  MoveL 662 to (32.13, 61.05, 0) mm, rotated rx -180 ry 0 rz -39.83 deg; joints [41.433, -75.782, 84.647, -0.866, 81.037, 41.564]
  MoveL 663 to (31.59, 62.21, 0) mm, rotated rx -180 ry 0 rz -39.83 deg; joints [41.415, -75.681, 84.52, -0.865, 81.064, 41.545]
  MoveL 664 to (31.21, 63.13, 0) mm, rotated rx 180 ry 0 rz -39.83 deg; joints [41.403, -75.601, 84.419, -0.865, 81.084, 41.533]
  MoveL 665 to (30.87, 64.05, 0) mm, rotated rx 180 ry 0 rz -39.83 deg; joints [41.392, -75.521, 84.319, -0.865, 81.105, 41.522]
  MoveL 666 to (30.56, 64.99, 0) mm, rotated rx -180 ry 0 rz -39.83 deg; joints [41.383, -75.441, 84.217, -0.865, 81.126, 41.513]
  MoveL 667 to (30.26, 65.94, 0) mm, rotated rx 180 ry 0 rz -39.83 deg; joints [41.376, -75.36, 84.115, -0.865, 81.148, 41.505]
  MoveL 668 to (30, 66.82, 0) mm, rotated rx 180 ry 0 rz -39.83 deg; joints [41.369, -75.285, 84.019, -0.865, 81.167, 41.498]
  MoveL 669 to (29.76, 67.7, 0) mm, rotated rx 180 ry 0 rz -39.83 deg; joints [41.364, -75.209, 83.924, -0.865, 81.188, 41.492]
  MoveL 670 to (29.54, 68.6, 0) mm, rotated rx 180 ry 0 rz -39.83 deg; joints [41.36, -75.134, 83.828, -0.865, 81.208, 41.488]
  MoveL 671 to (29.35, 69.49, 0) mm, rotated rx 180 ry 0 rz -39.83 deg; joints [41.357, -75.058, 83.732, -0.865, 81.228, 41.485]
  MoveL 672 to (29.18, 70.5, 0) mm, rotated rx 180 ry 0 rz -39.83 deg; joints [41.356, -74.974, 83.625, -0.865, 81.251, 41.484]
  MoveL 673 to (29.04, 71.51, 0) mm, rotated rx 180 ry 0 rz -39.83 deg; joints [41.357, -74.889, 83.518, -0.865, 81.274, 41.484]
  MoveL 674 to (28.93, 72.53, 0) mm, rotated rx 180 ry 0 rz -39.83 deg; joints [41.36, -74.805, 83.41, -0.865, 81.297, 41.487]
  MoveL 675 to (28.85, 73.55, 0) mm, rotated rx -180 ry 0 rz -39.83 deg; joints [41.364, -74.721, 83.303, -0.865, 81.32, 41.49]
  MoveL 676 to (28.8, 74.65, 0) mm, rotated rx 180 ry 0 rz -39.83 deg; joints [41.37, -74.63, 83.188, -0.865, 81.344, 41.496]
  MoveL 677 to (28.77, 75.75, 0) mm, rotated rx 180 ry 0 rz -39.83 deg; joints [41.377, -74.54, 83.073, -0.865, 81.369, 41.503]
  MoveL 678 to (28.79, 76.84, 0) mm, rotated rx 180 ry 0 rz -39.83 deg; joints [41.387, -74.45, 82.958, -0.865, 81.394, 41.512]
  MoveL 679 to (28.85, 77.94, 0) mm, rotated rx 180 ry 0 rz -39.83 deg; joints [41.399, -74.362, 82.845, -0.865, 81.419, 41.524]
  MoveL 680 to (28.94, 78.85, 0) mm, rotated rx 180 ry 0 rz -39.83 deg; joints [41.411, -74.288, 82.751, -0.865, 81.44, 41.535]
  MoveL 681 to (29.07, 79.77, 0) mm, rotated rx 180 ry 0 rz -39.83 deg; joints [41.424, -74.215, 82.657, -0.865, 81.46, 41.549]
  MoveL 682 to (29.23, 80.68, 0) mm, rotated rx 180 ry 0 rz -39.83 deg; joints [41.44, -74.142, 82.565, -0.865, 81.48, 41.564]
  MoveL 683 to (29.43, 81.58, 0) mm, rotated rx 180 ry 0 rz -39.83 deg; joints [41.457, -74.071, 82.473, -0.865, 81.501, 41.581]
  MoveL 684 to (29.67, 82.48, 0) mm, rotated rx 180 ry 0 rz -39.83 deg; joints [41.476, -74, 82.383, -0.865, 81.521, 41.6]
  MoveL 685 to (29.95, 83.36, 0) mm, rotated rx 180 ry 0 rz -39.83 deg; joints [41.498, -73.931, 82.294, -0.865, 81.54, 41.621]
  MoveL 686 to (30.28, 84.22, 0) mm, rotated rx -180 ry 0 rz -39.83 deg; joints [41.521, -73.864, 82.209, -0.865, 81.559, 41.644]
  MoveL 687 to (30.68, 85.06, 0) mm, rotated rx -180 ry 0 rz -39.83 deg; joints [41.548, -73.801, 82.128, -0.865, 81.577, 41.671]
  MoveL 688 to (30.93, 85.51, 0) mm, rotated rx 180 ry 0 rz -39.83 deg; joints [41.565, -73.767, 82.085, -0.865, 81.587, 41.687]
  MoveL 689 to (31.21, 85.95, 0) mm, rotated rx 180 ry 0 rz -39.83 deg; joints [41.582, -73.734, 82.043, -0.865, 81.596, 41.705]
  MoveL 690 to (31.51, 86.38, 0) mm, rotated rx 180 ry 0 rz -39.83 deg; joints [41.601, -73.703, 82.002, -0.865, 81.605, 41.723]
  MoveL 691 to (31.84, 86.79, 0) mm, rotated rx 180 ry 0 rz -39.83 deg; joints [41.621, -73.673, 81.964, -0.865, 81.614, 41.743]
  MoveL 692 to (32.24, 87.26, 0) mm, rotated rx 180 ry 0 rz -39.83 deg; joints [41.645, -73.639, 81.921, -0.865, 81.624, 41.767]
  MoveL 693 to (32.68, 87.7, 0) mm, rotated rx 180 ry 0 rz -39.83 deg; joints [41.671, -73.608, 81.882, -0.865, 81.632, 41.793]
  MoveL 694 to (33.15, 88.1, 0) mm, rotated rx 180 ry 0 rz -39.83 deg; joints [41.698, -73.581, 81.848, -0.865, 81.64, 41.82]
  MoveL 695 to (33.66, 88.45, 0) mm, rotated rx 180 ry 0 rz -39.83 deg; joints [41.726, -73.559, 81.819, -0.865, 81.646, 41.848]
  MoveL 696 to (33.98, 88.63, 0) mm, rotated rx 180 ry 0 rz -39.83 deg; joints [41.744, -73.547, 81.805, -0.865, 81.649, 41.866]
  MoveL 697 to (34.31, 88.8, 0) mm, rotated rx -180 ry 0 rz -39.83 deg; joints [41.762, -73.537, 81.793, -0.865, 81.652, 41.884]
  MoveL 698 to (34.64, 88.96, 0) mm, rotated rx 180 ry 0 rz -39.83 deg; joints [41.781, -73.528, 81.782, -0.865, 81.655, 41.902]
  MoveL 699 to (34.98, 89.11, 0) mm, rotated rx -180 ry 0 rz -39.83 deg; joints [41.799, -73.52, 81.771, -0.865, 81.657, 41.921]
  Establecer velocidad (1000.0 mm/s)
  MoveL 700 to (34.98, 89.11, 0) mm, rotated rx -180 ry 0 rz -39.83 deg; joints [41.799, -73.52, 81.771, -0.865, 81.657, 41.921]
  MoveL 701 to (34.98, 89.11, 20) mm, rotated rx 180 ry 0 rz -39.83 deg; joints [41.815, -73.829, 80.433, -0.862, 83.304, 41.911]

--- program P_ou_1 (robot KUKA KR 16 2) ---
  Suave(1)
  Establecer velocidad (1000.0 mm/s)
  Est. Ref.: Frame 2
  Est. herr: Plumon_ensamble
  Mostrar Plumon_ensamble
  MoveJ 1 to (24.64, 146.17, 20) mm, rotated rx 180 ry 0 rz -39.83 deg; joints [41.72, -68.932, 73.922, -0.859, 84.916, 41.792]
  MoveL 2 to (24.64, 146.17, 20) mm, rotated rx 180 ry 0 rz -39.83 deg; joints [41.72, -68.932, 73.922, -0.859, 84.916, 41.792]
  MoveL 3 to (24.64, 146.17, 0) mm, rotated rx -180 ry 0 rz -39.83 deg; joints [41.705, -68.665, 75.285, -0.861, 83.287, 41.802]
  MoveL 4 to (24.64, 146.17, 0) mm, rotated rx -180 ry 0 rz -39.83 deg; joints [41.705, -68.665, 75.285, -0.861, 83.287, 41.802]
  Establecer velocidad (50.0 mm/s)
  MoveL 5 to (24.63, 147.55, 0) mm, rotated rx 180 ry 0 rz -39.83 deg; joints [41.715, -68.548, 75.124, -0.861, 83.331, 41.811]
  MoveL 6 to (24.63, 148.94, 0) mm, rotated rx 180 ry 0 rz -39.83 deg; joints [41.724, -68.431, 74.964, -0.861, 83.375, 41.82]
  MoveL 7 to (24.65, 150.33, 0) mm, rotated rx -180 ry 0 rz -39.83 deg; joints [41.735, -68.315, 74.803, -0.861, 83.419, 41.83]
  MoveL 8 to (24.7, 151.72, 0) mm, rotated rx 180 ry 0 rz -39.83 deg; joints [41.748, -68.199, 74.643, -0.861, 83.463, 41.842]
  MoveL 9 to (24.78, 152.98, 0) mm, rotated rx 180 ry 0 rz -39.83 deg; joints [41.761, -68.093, 74.497, -0.861, 83.504, 41.854]
  MoveL 10 to (24.9, 154.25, 0) mm, rotated rx 180 ry 0 rz -39.83 deg; joints [41.775, -67.988, 74.352, -0.861, 83.544, 41.868]
  MoveL 11 to (25.06, 155.51, 0) mm, rotated rx 180 ry 0 rz -39.83 deg; joints [41.792, -67.884, 74.208, -0.861, 83.584, 41.884]
  MoveL 12 to (25.27, 156.76, 0) mm, rotated rx 180 ry 0 rz -39.83 deg; joints [41.811, -67.781, 74.065, -0.861, 83.624, 41.903]
  MoveL 13 to (25.55, 158.04, 0) mm, rotated rx 180 ry 0 rz -39.83 deg; joints [41.833, -67.676, 73.92, -0.861, 83.665, 41.924]
  MoveL 14 to (25.87, 159.31, 0) mm, rotated rx -180 ry 0 rz -39.83 deg; joints [41.858, -67.573, 73.777, -0.861, 83.705, 41.949]
  MoveL 15 to (26.26, 160.56, 0) mm, rotated rx 180 ry 0 rz -39.83 deg; joints [41.885, -67.472, 73.636, -0.861, 83.745, 41.975]
  MoveL 16 to (26.69, 161.8, 0) mm, rotated rx 180 ry 0 rz -39.83 deg; joints [41.915, -67.372, 73.498, -0.861, 83.784, 42.004]
  MoveL 17 to (27.31, 163.33, 0) mm, rotated rx 180 ry 0 rz -39.83 deg; joints [41.955, -67.25, 73.329, -0.861, 83.832, 42.043]
  MoveL 18 to (28, 164.83, 0) mm, rotated rx -180 ry 0 rz -39.83 deg; joints [41.998, -67.131, 73.163, -0.861, 83.879, 42.086]
  MoveL 19 to (28.74, 166.31, 0) mm, rotated rx -180 ry 0 rz -39.83 deg; joints [42.044, -67.014, 73, -0.861, 83.925, 42.131]
  MoveL 20 to (29.52, 167.78, 0) mm, rotated rx 180 ry 0 rz -39.83 deg; joints [42.091, -66.899, 72.84, -0.861, 83.971, 42.177]
  MoveL 21 to (30.17, 168.94, 0) mm, rotated rx -180 ry 0 rz -39.83 deg; joints [42.13, -66.807, 72.713, -0.861, 84.008, 42.216]
  MoveL 22 to (30.85, 170.09, 0) mm, rotated rx -180 ry 0 rz -39.83 deg; joints [42.17, -66.718, 72.588, -0.861, 84.043, 42.255]
  MoveL 23 to (31.58, 171.21, 0) mm, rotated rx 180 ry 0 rz -39.83 deg; joints [42.212, -66.631, 72.467, -0.861, 84.078, 42.297]
  MoveL 24 to (32.35, 172.28, 0) mm, rotated rx 180 ry 0 rz -39.83 deg; joints [42.256, -66.549, 72.352, -0.861, 84.111, 42.34]
  MoveL 25 to (33.37, 173.51, 0) mm, rotated rx 180 ry 0 rz -39.83 deg; joints [42.312, -66.456, 72.223, -0.861, 84.149, 42.396]
  MoveL 26 to (34.47, 174.67, 0) mm, rotated rx 180 ry 0 rz -39.83 deg; joints [42.372, -66.37, 72.103, -0.861, 84.184, 42.456]
  MoveL 27 to (35.63, 175.78, 0) mm, rotated rx 180 ry 0 rz -39.83 deg; joints [42.434, -66.288, 71.989, -0.861, 84.217, 42.517]
  MoveL 28 to (36.83, 176.85, 0) mm, rotated rx 180 ry 0 rz -39.83 deg; joints [42.498, -66.21, 71.88, -0.861, 84.248, 42.58]
  MoveL 29 to (38.25, 178.06, 0) mm, rotated rx 180 ry 0 rz -39.83 deg; joints [42.573, -66.123, 71.758, -0.861, 84.284, 42.655]
  MoveL 30 to (39.7, 179.21, 0) mm, rotated rx 180 ry 0 rz -39.83 deg; joints [42.649, -66.04, 71.643, -0.861, 84.317, 42.73]
  MoveL 31 to (41.21, 180.29, 0) mm, rotated rx 180 ry 0 rz -39.83 deg; joints [42.727, -65.964, 71.538, -0.861, 84.348, 42.808]
  MoveL 32 to (42.77, 181.27, 0) mm, rotated rx 180 ry 0 rz -39.83 deg; joints [42.807, -65.897, 71.445, -0.861, 84.375, 42.888]
  MoveL 33 to (43.73, 181.8, 0) mm, rotated rx -180 ry 0 rz -39.83 deg; joints [42.856, -65.863, 71.398, -0.861, 84.389, 42.936]
  MoveL 34 to (44.71, 182.29, 0) mm, rotated rx 180 ry 0 rz -39.83 deg; joints [42.905, -65.831, 71.354, -0.861, 84.402, 42.985]
  MoveL 35 to (45.7, 182.76, 0) mm, rotated rx 180 ry 0 rz -39.83 deg; joints [42.955, -65.801, 71.313, -0.861, 84.413, 43.035]
  MoveL 36 to (46.7, 183.22, 0) mm, rotated rx 180 ry 0 rz -39.83 deg; joints [43.005, -65.773, 71.274, -0.861, 84.425, 43.085]
  Establecer velocidad (1000.0 mm/s)
  MoveL 37 to (46.7, 183.22, 0) mm, rotated rx 180 ry 0 rz -39.83 deg; joints [43.005, -65.773, 71.274, -0.861, 84.425, 43.085]
  MoveL 38 to (46.7, 183.22, 20) mm, rotated rx 180 ry 0 rz -39.83 deg; joints [43.019, -66.01, 69.886, -0.859, 86.049, 43.074]
  Establecer velocidad (1000.0 mm/s)
  MoveL 39 to (24.64, 146.17, 20) mm, rotated rx 180 ry 0 rz -39.83 deg; joints [41.72, -68.932, 73.922, -0.859, 84.916, 41.792]
  MoveL 40 to (24.64, 146.17, 0) mm, rotated rx -180 ry 0 rz -39.83 deg; joints [41.705, -68.665, 75.285, -0.861, 83.287, 41.802]
  MoveL 41 to (24.64, 146.17, 0) mm, rotated rx -180 ry 0 rz -39.83 deg; joints [41.705, -68.665, 75.285, -0.861, 83.287, 41.802]
  Establecer velocidad (50.0 mm/s)
  MoveL 42 to (24.43, 145.76, 0) mm, rotated rx 180 ry 0 rz -39.83 deg; joints [41.692, -68.696, 75.328, -0.861, 83.275, 41.789]
  MoveL 43 to (24.21, 145.35, 0) mm, rotated rx 180 ry 0 rz -39.83 deg; joints [41.678, -68.728, 75.371, -0.861, 83.263, 41.776]
  MoveL 44 to (24.01, 144.94, 0) mm, rotated rx 180 ry 0 rz -39.83 deg; joints [41.666, -68.76, 75.415, -0.861, 83.252, 41.763]
  MoveL 45 to (23.83, 144.52, 0) mm, rotated rx 180 ry 0 rz -39.83 deg; joints [41.654, -68.793, 75.46, -0.861, 83.239, 41.751]
  MoveL 46 to (23.64, 144.02, 0) mm, rotated rx 180 ry 0 rz -39.83 deg; joints [41.641, -68.833, 75.513, -0.861, 83.225, 41.738]
  MoveL 47 to (23.47, 143.51, 0) mm, rotated rx 180 ry 0 rz -39.83 deg; joints [41.629, -68.873, 75.569, -0.861, 83.21, 41.727]
  MoveL 48 to (23.32, 143, 0) mm, rotated rx -180 ry 0 rz -39.83 deg; joints [41.618, -68.914, 75.625, -0.861, 83.195, 41.716]
  MoveL 49 to (23.17, 142.49, 0) mm, rotated rx 180 ry 0 rz -39.83 deg; joints [41.607, -68.955, 75.681, -0.861, 83.18, 41.705]
  MoveL 50 to (23.17, 142.49, 0) mm, rotated rx 180 ry 0 rz -39.83 deg; joints [41.607, -68.955, 75.681, -0.861, 83.18, 41.705]
  MoveL 51 to (22.09, 141.81, 0) mm, rotated rx -180 ry 0 rz -39.83 deg; joints [41.549, -68.998, 75.739, -0.861, 83.164, 41.648]
  MoveL 52 to (21.01, 141.12, 0) mm, rotated rx 180 ry 0 rz -39.83 deg; joints [41.492, -69.043, 75.798, -0.861, 83.149, 41.591]
  MoveL 53 to (19.96, 140.4, 0) mm, rotated rx 180 ry 0 rz -39.83 deg; joints [41.435, -69.09, 75.86, -0.861, 83.132, 41.534]
  MoveL 54 to (18.94, 139.64, 0) mm, rotated rx 180 ry 0 rz -39.83 deg; joints [41.38, -69.14, 75.928, -0.861, 83.114, 41.479]
  MoveL 55 to (17.59, 138.51, 0) mm, rotated rx 180 ry 0 rz -39.83 deg; joints [41.306, -69.218, 76.032, -0.861, 83.086, 41.405]
  MoveL 56 to (16.32, 137.28, 0) mm, rotated rx 180 ry 0 rz -39.83 deg; joints [41.234, -69.304, 76.149, -0.861, 83.055, 41.335]
  MoveL 57 to (15.13, 135.97, 0) mm, rotated rx 180 ry 0 rz -39.83 deg; joints [41.166, -69.398, 76.275, -0.861, 83.022, 41.267]
  MoveL 58 to (14.03, 134.58, 0) mm, rotated rx 180 ry 0 rz -39.83 deg; joints [41.102, -69.499, 76.411, -0.861, 82.986, 41.203]
  MoveL 59 to (13.16, 133.37, 0) mm, rotated rx 180 ry 0 rz -39.83 deg; joints [41.05, -69.589, 76.531, -0.861, 82.954, 41.152]
  MoveL 60 to (12.35, 132.13, 0) mm, rotated rx 180 ry 0 rz -39.83 deg; joints [41.001, -69.682, 76.657, -0.861, 82.921, 41.103]
  MoveL 61 to (11.59, 130.85, 0) mm, rotated rx 180 ry 0 rz -39.83 deg; joints [40.953, -69.778, 76.786, -0.861, 82.887, 41.056]
  MoveL 62 to (10.87, 129.55, 0) mm, rotated rx -180 ry 0 rz -39.83 deg; joints [40.908, -69.877, 76.919, -0.861, 82.853, 41.011]
  MoveL 63 to (10.02, 127.88, 0) mm, rotated rx -180 ry 0 rz -39.83 deg; joints [40.853, -70.004, 77.09, -0.861, 82.808, 40.956]
  MoveL 64 to (9.24, 126.19, 0) mm, rotated rx 180 ry 0 rz -39.83 deg; joints [40.801, -70.134, 77.265, -0.861, 82.763, 40.905]
  MoveL 65 to (8.56, 124.46, 0) mm, rotated rx 180 ry 0 rz -39.83 deg; joints [40.753, -70.269, 77.445, -0.861, 82.716, 40.858]
  MoveL 66 to (7.98, 122.69, 0) mm, rotated rx -180 ry 0 rz -39.83 deg; joints [40.71, -70.407, 77.631, -0.861, 82.668, 40.816]
  MoveL 67 to (7.57, 121.14, 0) mm, rotated rx 180 ry 0 rz -39.83 deg; joints [40.677, -70.53, 77.796, -0.861, 82.626, 40.784]
  MoveL 68 to (7.24, 119.56, 0) mm, rotated rx 180 ry 0 rz -39.83 deg; joints [40.648, -70.656, 77.964, -0.861, 82.583, 40.755]
  MoveL 69 to (6.97, 117.98, 0) mm, rotated rx -180 ry 0 rz -39.83 deg; joints [40.622, -70.784, 78.135, -0.861, 82.54, 40.73]
  MoveL 70 to (6.77, 116.38, 0) mm, rotated rx 180 ry 0 rz -39.83 deg; joints [40.598, -70.913, 78.308, -0.861, 82.496, 40.707]
  MoveL 71 to (6.61, 114.86, 0) mm, rotated rx 180 ry 0 rz -39.83 deg; joints [40.578, -71.036, 78.472, -0.861, 82.454, 40.687]
  MoveL 72 to (6.51, 113.35, 0) mm, rotated rx 180 ry 0 rz -39.83 deg; joints [40.56, -71.16, 78.637, -0.861, 82.413, 40.67]
  MoveL 73 to (6.47, 111.83, 0) mm, rotated rx -180 ry 0 rz -39.83 deg; joints [40.545, -71.285, 78.803, -0.861, 82.372, 40.655]
  MoveL 74 to (6.5, 110.32, 0) mm, rotated rx 180 ry 0 rz -39.83 deg; joints [40.534, -71.41, 78.969, -0.861, 82.33, 40.645]
  MoveL 75 to (6.61, 108.85, 0) mm, rotated rx 180 ry 0 rz -39.83 deg; joints [40.527, -71.533, 79.132, -0.861, 82.29, 40.638]
  MoveL 76 to (6.78, 107.39, 0) mm, rotated rx 180 ry 0 rz -39.83 deg; joints [40.523, -71.656, 79.295, -0.861, 82.25, 40.635]
  MoveL 77 to (7.02, 105.93, 0) mm, rotated rx -180 ry 0 rz -39.83 deg; joints [40.523, -71.779, 79.459, -0.861, 82.209, 40.636]
  MoveL 78 to (7.3, 104.48, 0) mm, rotated rx 180 ry 0 rz -39.83 deg; joints [40.525, -71.903, 79.622, -0.861, 82.17, 40.638]
  MoveL 79 to (7.53, 103.44, 0) mm, rotated rx -180 ry 0 rz -39.83 deg; joints [40.527, -71.991, 79.74, -0.861, 82.141, 40.641]
  MoveL 80 to (7.78, 102.4, 0) mm, rotated rx 180 ry 0 rz -39.83 deg; joints [40.531, -72.08, 79.857, -0.862, 82.112, 40.645]
  MoveL 81 to (8.06, 101.38, 0) mm, rotated rx 180 ry 0 rz -39.83 deg; joints [40.536, -72.168, 79.973, -0.862, 82.084, 40.651]
  MoveL 82 to (8.38, 100.36, 0) mm, rotated rx -180 ry 0 rz -39.83 deg; joints [40.543, -72.256, 80.089, -0.862, 82.056, 40.658]
  MoveL 83 to (8.85, 99.02, 0) mm, rotated rx 180 ry 0 rz -39.83 deg; joints [40.556, -72.372, 80.243, -0.862, 82.02, 40.671]
  MoveL 84 to (9.39, 97.71, 0) mm, rotated rx -180 ry 0 rz -39.83 deg; joints [40.571, -72.488, 80.395, -0.862, 81.983, 40.688]
  MoveL 85 to (9.97, 96.41, 0) mm, rotated rx 180 ry 0 rz -39.83 deg; joints [40.59, -72.603, 80.546, -0.862, 81.947, 40.707]
  MoveL 86 to (10.6, 95.12, 0) mm, rotated rx 180 ry 0 rz -39.83 deg; joints [40.61, -72.716, 80.695, -0.862, 81.912, 40.728]
  MoveL 87 to (11.22, 93.91, 0) mm, rotated rx 180 ry 0 rz -39.83 deg; joints [40.632, -72.824, 80.837, -0.862, 81.878, 40.75]
  MoveL 88 to (11.9, 92.73, 0) mm, rotated rx 180 ry 0 rz -39.83 deg; joints [40.656, -72.93, 80.976, -0.862, 81.846, 40.774]
  MoveL 89 to (12.62, 91.59, 0) mm, rotated rx 180 ry 0 rz -39.83 deg; joints [40.683, -73.034, 81.112, -0.862, 81.814, 40.802]
  MoveL 90 to (13.42, 90.49, 0) mm, rotated rx 180 ry 0 rz -39.83 deg; joints [40.714, -73.135, 81.243, -0.863, 81.783, 40.833]
  MoveL 91 to (14.09, 89.67, 0) mm, rotated rx 180 ry 0 rz -39.83 deg; joints [40.741, -73.211, 81.343, -0.863, 81.76, 40.861]
  MoveL 92 to (14.81, 88.88, 0) mm, rotated rx 180 ry 0 rz -39.83 deg; joints [40.771, -73.285, 81.44, -0.863, 81.737, 40.891]
  MoveL 93 to (15.55, 88.11, 0) mm, rotated rx 180 ry 0 rz -39.83 deg; joints [40.802, -73.358, 81.536, -0.863, 81.715, 40.922]
  MoveL 94 to (16.3, 87.35, 0) mm, rotated rx 180 ry 0 rz -39.83 deg; joints [40.833, -73.43, 81.63, -0.863, 81.694, 40.954]
  MoveL 95 to (16.3, 87.35, 0) mm, rotated rx 180 ry 0 rz -39.83 deg; joints [40.833, -73.43, 81.63, -0.863, 81.694, 40.954]
  MoveL 96 to (16.8, 85.15, 0) mm, rotated rx 180 ry 0 rz -39.83 deg; joints [40.841, -73.617, 81.872, -0.863, 81.638, 40.962]
  MoveL 97 to (17.32, 82.96, 0) mm, rotated rx -180 ry 0 rz -39.83 deg; joints [40.849, -73.803, 82.113, -0.863, 81.584, 40.971]
  MoveL 98 to (17.9, 80.78, 0) mm, rotated rx 180 ry 0 rz -39.83 deg; joints [40.86, -73.989, 82.353, -0.863, 81.53, 40.983]
  MoveL 99 to (18.54, 78.63, 0) mm, rotated rx 180 ry 0 rz -39.83 deg; joints [40.875, -74.174, 82.591, -0.864, 81.477, 40.999]
  MoveL 100 to (19.22, 76.65, 0) mm, rotated rx 180 ry 0 rz -39.83 deg; joints [40.893, -74.345, 82.811, -0.864, 81.429, 41.018]
  MoveL 101 to (19.97, 74.68, 0) mm, rotated rx 180 ry 0 rz -39.83 deg; joints [40.915, -74.515, 83.029, -0.864, 81.381, 41.04]
  MoveL 102 to (20.75, 72.73, 0) mm, rotated rx 180 ry 0 rz -39.83 deg; joints [40.939, -74.684, 83.246, -0.864, 81.334, 41.065]
  MoveL 103 to (21.56, 70.79, 0) mm, rotated rx 180 ry 0 rz -39.83 deg; joints [40.964, -74.854, 83.462, -0.864, 81.287, 41.091]
  MoveL 104 to (21.56, 70.79, 0) mm, rotated rx 180 ry 0 rz -39.83 deg; joints [40.964, -74.854, 83.462, -0.864, 81.287, 41.091]
  MoveL 105 to (22.1, 68.18, 0) mm, rotated rx 180 ry 0 rz -39.83 deg; joints [40.971, -75.074, 83.742, -0.864, 81.228, 41.098]
  MoveL 106 to (22.69, 65.58, 0) mm, rotated rx -180 ry 0 rz -39.83 deg; joints [40.979, -75.294, 84.021, -0.864, 81.169, 41.108]
  MoveL 107 to (23.37, 63, 0) mm, rotated rx 180 ry 0 rz -39.83 deg; joints [40.993, -75.512, 84.297, -0.865, 81.111, 41.122]
  MoveL 108 to (24.17, 60.46, 0) mm, rotated rx 180 ry 0 rz -39.83 deg; joints [41.013, -75.729, 84.571, -0.865, 81.055, 41.144]
  MoveL 109 to (24.64, 59.19, 0) mm, rotated rx -180 ry 0 rz -39.83 deg; joints [41.027, -75.839, 84.709, -0.865, 81.027, 41.158]
  MoveL 110 to (25.16, 57.94, 0) mm, rotated rx 180 ry 0 rz -39.83 deg; joints [41.044, -75.948, 84.846, -0.865, 80.999, 41.175]
  MoveL 111 to (25.74, 56.72, 0) mm, rotated rx 180 ry 0 rz -39.83 deg; joints [41.064, -76.055, 84.98, -0.865, 80.972, 41.196]
  MoveL 112 to (26.38, 55.53, 0) mm, rotated rx -180 ry 0 rz -39.83 deg; joints [41.088, -76.16, 85.112, -0.865, 80.945, 41.22]
  MoveL 113 to (27.01, 54.5, 0) mm, rotated rx 180 ry 0 rz -39.83 deg; joints [41.112, -76.252, 85.228, -0.865, 80.922, 41.245]
  MoveL 114 to (27.68, 53.5, 0) mm, rotated rx 180 ry 0 rz -39.83 deg; joints [41.139, -76.342, 85.341, -0.865, 80.899, 41.272]
  MoveL 115 to (28.39, 52.51, 0) mm, rotated rx 180 ry 0 rz -39.83 deg; joints [41.168, -76.431, 85.453, -0.866, 80.877, 41.301]
  MoveL 116 to (29.11, 51.54, 0) mm, rotated rx 180 ry 0 rz -39.83 deg; joints [41.197, -76.52, 85.564, -0.866, 80.855, 41.331]
  MoveL 117 to (29.89, 50.49, 0) mm, rotated rx 180 ry 0 rz -39.83 deg; joints [41.23, -76.614, 85.682, -0.866, 80.832, 41.364]
  MoveL 118 to (30.7, 49.47, 0) mm, rotated rx -180 ry 0 rz -39.83 deg; joints [41.264, -76.708, 85.799, -0.866, 80.809, 41.398]
  MoveL 119 to (31.53, 48.46, 0) mm, rotated rx 180 ry 0 rz -39.83 deg; joints [41.299, -76.8, 85.914, -0.866, 80.787, 41.434]
  MoveL 120 to (32.39, 47.49, 0) mm, rotated rx 180 ry 0 rz -39.83 deg; joints [41.337, -76.891, 86.027, -0.866, 80.765, 41.472]
  MoveL 121 to (33.11, 46.72, 0) mm, rotated rx 180 ry 0 rz -39.83 deg; joints [41.369, -76.962, 86.116, -0.866, 80.748, 41.504]
  MoveL 122 to (33.87, 45.98, 0) mm, rotated rx -180 ry 0 rz -39.83 deg; joints [41.403, -77.031, 86.202, -0.866, 80.731, 41.539]
  MoveL 123 to (34.65, 45.27, 0) mm, rotated rx -180 ry 0 rz -39.83 deg; joints [41.439, -77.098, 86.286, -0.866, 80.715, 41.574]
  MoveL 124 to (35.45, 44.59, 0) mm, rotated rx 180 ry 0 rz -39.83 deg; joints [41.476, -77.164, 86.368, -0.866, 80.7, 41.612]
  MoveL 125 to (36.39, 43.86, 0) mm, rotated rx 180 ry 0 rz -39.83 deg; joints [41.52, -77.235, 86.456, -0.867, 80.683, 41.656]
  MoveL 126 to (37.35, 43.16, 0) mm, rotated rx -180 ry 0 rz -39.83 deg; joints [41.565, -77.303, 86.542, -0.867, 80.667, 41.702]
  MoveL 127 to (38.33, 42.49, 0) mm, rotated rx 180 ry 0 rz -39.83 deg; joints [41.612, -77.37, 86.625, -0.867, 80.651, 41.749]
  MoveL 128 to (39.32, 41.83, 0) mm, rotated rx 180 ry 0 rz -39.83 deg; joints [41.659, -77.435, 86.706, -0.867, 80.635, 41.797]
  MoveL 129 to (40.09, 41.34, 0) mm, rotated rx 180 ry 0 rz -39.83 deg; joints [41.696, -77.484, 86.767, -0.867, 80.624, 41.834]
  MoveL 130 to (40.86, 40.86, 0) mm, rotated rx -180 ry 0 rz -39.83 deg; joints [41.733, -77.533, 86.827, -0.867, 80.613, 41.871]
  MoveL 131 to (41.64, 40.4, 0) mm, rotated rx 180 ry 0 rz -39.83 deg; joints [41.771, -77.579, 86.886, -0.867, 80.602, 41.909]
  MoveL 132 to (42.43, 39.96, 0) mm, rotated rx -180 ry 0 rz -39.83 deg; joints [41.81, -77.624, 86.942, -0.867, 80.591, 41.948]
  MoveL 133 to (43.59, 39.38, 0) mm, rotated rx 180 ry 0 rz -39.83 deg; joints [41.867, -77.685, 87.017, -0.867, 80.577, 42.006]
  MoveL 134 to (44.76, 38.84, 0) mm, rotated rx 180 ry 0 rz -39.83 deg; joints [41.926, -77.743, 87.089, -0.868, 80.564, 42.065]
  MoveL 135 to (45.96, 38.33, 0) mm, rotated rx 180 ry 0 rz -39.83 deg; joints [41.986, -77.798, 87.158, -0.868, 80.551, 42.125]
  MoveL 136 to (47.15, 37.83, 0) mm, rotated rx 180 ry 0 rz -39.83 deg; joints [42.047, -77.852, 87.226, -0.868, 80.539, 42.185]
  MoveL 137 to (47.15, 37.83, 0) mm, rotated rx 180 ry 0 rz -39.83 deg; joints [42.047, -77.852, 87.226, -0.868, 80.539, 42.185]
  MoveL 138 to (48.32, 36.91, 0) mm, rotated rx 180 ry 0 rz -39.83 deg; joints [42.102, -77.941, 87.335, -0.868, 80.519, 42.241]
  MoveL 139 to (49.49, 35.99, 0) mm, rotated rx 180 ry 0 rz -39.83 deg; joints [42.158, -78.029, 87.443, -0.868, 80.499, 42.297]
  MoveL 140 to (50.68, 35.09, 0) mm, rotated rx -180 ry 0 rz -39.83 deg; joints [42.215, -78.115, 87.55, -0.868, 80.48, 42.355]
  MoveL 141 to (51.89, 34.23, 0) mm, rotated rx -180 ry 0 rz -39.83 deg; joints [42.273, -78.199, 87.653, -0.868, 80.461, 42.413]
  MoveL 142 to (52.71, 33.66, 0) mm, rotated rx 180 ry 0 rz -39.83 deg; joints [42.314, -78.254, 87.721, -0.868, 80.449, 42.454]
  MoveL 143 to (53.55, 33.11, 0) mm, rotated rx 180 ry 0 rz -39.83 deg; joints [42.355, -78.308, 87.788, -0.869, 80.437, 42.495]
  MoveL 144 to (54.4, 32.58, 0) mm, rotated rx -180 ry 0 rz -39.83 deg; joints [42.397, -78.361, 87.853, -0.869, 80.426, 42.537]
  MoveL 145 to (55.26, 32.05, 0) mm, rotated rx 180 ry 0 rz -39.83 deg; joints [42.439, -78.413, 87.917, -0.869, 80.414, 42.58]
  MoveL 146 to (56.32, 31.41, 0) mm, rotated rx -180 ry 0 rz -39.83 deg; joints [42.492, -78.477, 87.995, -0.869, 80.401, 42.633]
  MoveL 147 to (57.4, 30.78, 0) mm, rotated rx 180 ry 0 rz -39.83 deg; joints [42.545, -78.54, 88.072, -0.869, 80.387, 42.686]
  MoveL 148 to (58.48, 30.17, 0) mm, rotated rx 180 ry 0 rz -39.83 deg; joints [42.599, -78.601, 88.148, -0.869, 80.374, 42.741]
  MoveL 149 to (59.57, 29.58, 0) mm, rotated rx 180 ry 0 rz -39.83 deg; joints [42.654, -78.661, 88.221, -0.869, 80.361, 42.796]
  MoveL 150 to (60.92, 28.87, 0) mm, rotated rx -180 ry 0 rz -39.83 deg; joints [42.723, -78.732, 88.309, -0.869, 80.346, 42.865]
  MoveL 151 to (62.29, 28.2, 0) mm, rotated rx 180 ry 0 rz -39.83 deg; joints [42.792, -78.802, 88.394, -0.869, 80.331, 42.934]
  MoveL 152 to (63.68, 27.55, 0) mm, rotated rx 180 ry 0 rz -39.83 deg; joints [42.863, -78.869, 88.476, -0.87, 80.317, 43.005]
  MoveL 153 to (65.07, 26.93, 0) mm, rotated rx 180 ry 0 rz -39.83 deg; joints [42.934, -78.933, 88.556, -0.87, 80.303, 43.077]
  MoveL 154 to (66.63, 26.27, 0) mm, rotated rx -180 ry 0 rz -39.83 deg; joints [43.015, -79.003, 88.641, -0.87, 80.289, 43.158]
  MoveL 155 to (68.2, 25.64, 0) mm, rotated rx 180 ry 0 rz -39.83 deg; joints [43.096, -79.07, 88.724, -0.87, 80.274, 43.239]
  MoveL 156 to (69.78, 25.02, 0) mm, rotated rx 180 ry 0 rz -39.83 deg; joints [43.177, -79.136, 88.805, -0.87, 80.261, 43.321]
  MoveL 157 to (71.36, 24.41, 0) mm, rotated rx 180 ry 0 rz -39.83 deg; joints [43.259, -79.201, 88.885, -0.87, 80.247, 43.403]
  MoveL 158 to (71.36, 24.41, 0) mm, rotated rx 180 ry 0 rz -39.83 deg; joints [43.259, -79.201, 88.885, -0.87, 80.247, 43.403]
  MoveL 159 to (71.89, 23.71, 0) mm, rotated rx -180 ry 0 rz -39.83 deg; joints [43.284, -79.264, 88.96, -0.87, 80.235, 43.428]
  MoveL 160 to (72.42, 23.01, 0) mm, rotated rx 180 ry 0 rz -39.83 deg; joints [43.309, -79.326, 89.034, -0.87, 80.222, 43.453]
  MoveL 161 to (72.98, 22.34, 0) mm, rotated rx 180 ry 0 rz -39.83 deg; joints [43.335, -79.386, 89.107, -0.87, 80.211, 43.479]
  MoveL 162 to (73.57, 21.7, 0) mm, rotated rx 180 ry 0 rz -39.83 deg; joints [43.363, -79.444, 89.177, -0.871, 80.199, 43.507]
  MoveL 163 to (74.45, 20.85, 0) mm, rotated rx 180 ry 0 rz -39.83 deg; joints [43.406, -79.521, 89.27, -0.871, 80.184, 43.55]
  MoveL 164 to (75.39, 20.07, 0) mm, rotated rx 180 ry 0 rz -39.83 deg; joints [43.452, -79.594, 89.357, -0.871, 80.17, 43.597]
  MoveL 165 to (76.37, 19.33, 0) mm, rotated rx 180 ry 0 rz -39.83 deg; joints [43.501, -79.663, 89.441, -0.871, 80.156, 43.646]
  MoveL 166 to (77.37, 18.62, 0) mm, rotated rx 180 ry 0 rz -39.83 deg; joints [43.551, -79.731, 89.522, -0.871, 80.143, 43.697]
  MoveL 167 to (78.43, 17.9, 0) mm, rotated rx 180 ry 0 rz -39.83 deg; joints [43.605, -79.8, 89.605, -0.871, 80.13, 43.75]
  MoveL 168 to (79.49, 17.19, 0) mm, rotated rx -180 ry 0 rz -39.83 deg; joints [43.658, -79.867, 89.686, -0.871, 80.117, 43.804]
  MoveL 169 to (80.56, 16.5, 0) mm, rotated rx 180 ry 0 rz -39.83 deg; joints [43.713, -79.933, 89.765, -0.871, 80.105, 43.859]
  MoveL 170 to (81.65, 15.85, 0) mm, rotated rx 180 ry 0 rz -39.83 deg; joints [43.769, -79.996, 89.842, -0.871, 80.093, 43.915]
  MoveL 171 to (82.83, 15.18, 0) mm, rotated rx -180 ry 0 rz -39.83 deg; joints [43.83, -80.061, 89.92, -0.871, 80.08, 43.977]
  MoveL 172 to (84.04, 14.56, 0) mm, rotated rx 180 ry 0 rz -39.83 deg; joints [43.893, -80.123, 89.994, -0.872, 80.069, 44.04]
  MoveL 173 to (85.27, 13.98, 0) mm, rotated rx -180 ry 0 rz -39.83 deg; joints [43.958, -80.18, 90.064, -0.872, 80.058, 44.104]
  MoveL 174 to (86.52, 13.46, 0) mm, rotated rx -180 ry 0 rz -39.83 deg; joints [44.024, -80.234, 90.128, -0.872, 80.048, 44.171]
  MoveL 175 to (87.55, 13.07, 0) mm, rotated rx 180 ry 0 rz -39.83 deg; joints [44.078, -80.274, 90.177, -0.872, 80.04, 44.226]
  MoveL 176 to (88.59, 12.73, 0) mm, rotated rx -180 ry 0 rz -39.83 deg; joints [44.134, -80.311, 90.222, -0.872, 80.033, 44.281]
  MoveL 177 to (89.64, 12.42, 0) mm, rotated rx 180 ry 0 rz -39.83 deg; joints [44.191, -80.346, 90.263, -0.872, 80.027, 44.338]
  MoveL 178 to (90.7, 12.13, 0) mm, rotated rx 180 ry 0 rz -39.83 deg; joints [44.248, -80.377, 90.302, -0.872, 80.02, 44.395]
  MoveL 179 to (91.93, 11.85, 0) mm, rotated rx -180 ry 0 rz -39.83 deg; joints [44.314, -80.411, 90.343, -0.872, 80.014, 44.462]
  MoveL 180 to (93.17, 11.59, 0) mm, rotated rx 180 ry 0 rz -39.83 deg; joints [44.382, -80.442, 90.381, -0.872, 80.008, 44.529]
  MoveL 181 to (94.41, 11.38, 0) mm, rotated rx 180 ry 0 rz -39.83 deg; joints [44.449, -80.469, 90.415, -0.872, 80.003, 44.597]
  MoveL 182 to (95.66, 11.19, 0) mm, rotated rx 180 ry 0 rz -39.83 deg; joints [44.518, -80.494, 90.445, -0.872, 79.998, 44.666]
  MoveL 183 to (96.8, 11.06, 0) mm, rotated rx 180 ry 0 rz -39.83 deg; joints [44.58, -80.514, 90.47, -0.872, 79.994, 44.728]
  MoveL 184 to (97.94, 10.95, 0) mm, rotated rx 180 ry 0 rz -39.83 deg; joints [44.643, -80.532, 90.492, -0.872, 79.99, 44.791]
  MoveL 185 to (99.09, 10.88, 0) mm, rotated rx 180 ry 0 rz -39.83 deg; joints [44.706, -80.546, 90.511, -0.873, 79.987, 44.855]
  MoveL 186 to (100.23, 10.85, 0) mm, rotated rx 180 ry 0 rz -39.83 deg; joints [44.77, -80.557, 90.525, -0.873, 79.985, 44.918]
  MoveL 187 to (100.6, 10.85, 0) mm, rotated rx 180 ry 0 rz -39.83 deg; joints [44.79, -80.56, 90.529, -0.873, 79.984, 44.939]
  MoveL 188 to (100.96, 10.86, 0) mm, rotated rx 180 ry 0 rz -39.83 deg; joints [44.811, -80.562, 90.532, -0.873, 79.984, 44.959]
  MoveL 189 to (101.33, 10.87, 0) mm, rotated rx -180 ry 0 rz -39.83 deg; joints [44.831, -80.564, 90.535, -0.873, 79.983, 44.979]
  MoveL 190 to (101.69, 10.88, 0) mm, rotated rx 180 ry 0 rz -39.83 deg; joints [44.851, -80.565, 90.537, -0.873, 79.983, 45]
  MoveL 191 to (101.69, 10.88, 0) mm, rotated rx 180 ry 0 rz -39.83 deg; joints [44.851, -80.565, 90.537, -0.873, 79.983, 45]
  MoveL 192 to (102.06, 10.87, 0) mm, rotated rx 180 ry 0 rz -39.83 deg; joints [44.872, -80.569, 90.542, -0.873, 79.982, 45.02]
  MoveL 193 to (102.43, 10.86, 0) mm, rotated rx 180 ry 0 rz -39.83 deg; joints [44.892, -80.573, 90.546, -0.873, 79.981, 45.04]
  MoveL 194 to (102.79, 10.85, 0) mm, rotated rx 180 ry 0 rz -39.83 deg; joints [44.912, -80.576, 90.55, -0.873, 79.98, 45.061]
  MoveL 195 to (103.16, 10.85, 0) mm, rotated rx 180 ry 0 rz -39.83 deg; joints [44.933, -80.578, 90.554, -0.873, 79.98, 45.081]
  MoveL 196 to (104.3, 10.88, 0) mm, rotated rx 180 ry 0 rz -39.83 deg; joints [44.997, -80.584, 90.562, -0.873, 79.978, 45.145]
  MoveL 197 to (105.45, 10.95, 0) mm, rotated rx -180 ry 0 rz -39.83 deg; joints [45.061, -80.587, 90.567, -0.873, 79.977, 45.209]
  MoveL 198 to (106.59, 11.06, 0) mm, rotated rx 180 ry 0 rz -39.83 deg; joints [45.125, -80.586, 90.568, -0.873, 79.977, 45.273]
  MoveL 199 to (107.73, 11.19, 0) mm, rotated rx 180 ry 0 rz -39.83 deg; joints [45.189, -80.583, 90.565, -0.873, 79.977, 45.337]
  MoveL 200 to (108.98, 11.38, 0) mm, rotated rx -180 ry 0 rz -39.83 deg; joints [45.259, -80.576, 90.559, -0.873, 79.977, 45.408]
  MoveL 201 to (110.22, 11.59, 0) mm, rotated rx 180 ry 0 rz -39.83 deg; joints [45.33, -80.567, 90.55, -0.873, 79.978, 45.478]
  MoveL 202 to (111.46, 11.85, 0) mm, rotated rx -180 ry 0 rz -39.83 deg; joints [45.4, -80.554, 90.537, -0.873, 79.98, 45.548]
  MoveL 203 to (112.68, 12.13, 0) mm, rotated rx 180 ry 0 rz -39.83 deg; joints [45.469, -80.539, 90.52, -0.873, 79.982, 45.618]
  MoveL 204 to (113.75, 12.42, 0) mm, rotated rx 180 ry 0 rz -39.83 deg; joints [45.53, -80.522, 90.502, -0.873, 79.984, 45.678]
  MoveL 205 to (114.8, 12.73, 0) mm, rotated rx 180 ry 0 rz -39.83 deg; joints [45.59, -80.503, 90.482, -0.873, 79.987, 45.738]
  MoveL 206 to (115.84, 13.07, 0) mm, rotated rx 180 ry 0 rz -39.83 deg; joints [45.649, -80.482, 90.457, -0.873, 79.99, 45.798]
  MoveL 207 to (116.87, 13.46, 0) mm, rotated rx 180 ry 0 rz -39.83 deg; joints [45.708, -80.457, 90.429, -0.873, 79.994, 45.856]
  MoveL 208 to (118.12, 13.98, 0) mm, rotated rx 180 ry 0 rz -39.83 deg; joints [45.78, -80.421, 90.39, -0.873, 80, 45.928]
  MoveL 209 to (119.35, 14.56, 0) mm, rotated rx 180 ry 0 rz -39.83 deg; joints [45.851, -80.381, 90.344, -0.873, 80.006, 45.999]
  MoveL 210 to (120.56, 15.18, 0) mm, rotated rx 180 ry 0 rz -39.83 deg; joints [45.921, -80.337, 90.294, -0.873, 80.013, 46.069]
  MoveL 211 to (121.74, 15.85, 0) mm, rotated rx 180 ry 0 rz -39.83 deg; joints [45.989, -80.289, 90.24, -0.873, 80.021, 46.137]
  MoveL 212 to (122.83, 16.5, 0) mm, rotated rx -180 ry 0 rz -39.83 deg; joints [46.052, -80.242, 90.185, -0.873, 80.029, 46.2]
  MoveL 213 to (123.9, 17.19, 0) mm, rotated rx 180 ry 0 rz -39.83 deg; joints [46.114, -80.191, 90.127, -0.873, 80.037, 46.262]
  MoveL 214 to (124.96, 17.9, 0) mm, rotated rx 180 ry 0 rz -39.83 deg; joints [46.176, -80.139, 90.067, -0.873, 80.046, 46.324]
  MoveL 215 to (126.01, 18.62, 0) mm, rotated rx -180 ry 0 rz -39.83 deg; joints [46.237, -80.085, 90.005, -0.873, 80.055, 46.384]
  MoveL 216 to (127.02, 19.33, 0) mm, rotated rx -180 ry 0 rz -39.83 deg; joints [46.295, -80.032, 89.944, -0.873, 80.064, 46.443]
  MoveL 217 to (128, 20.07, 0) mm, rotated rx -180 ry 0 rz -39.83 deg; joints [46.352, -79.977, 89.88, -0.873, 80.074, 46.499]
  MoveL 218 to (128.94, 20.85, 0) mm, rotated rx 180 ry 0 rz -39.83 deg; joints [46.407, -79.917, 89.811, -0.873, 80.084, 46.554]
  MoveL 219 to (129.82, 21.7, 0) mm, rotated rx 180 ry 0 rz -39.83 deg; joints [46.459, -79.853, 89.736, -0.873, 80.095, 46.606]
  MoveL 220 to (130.4, 22.34, 0) mm, rotated rx 180 ry 0 rz -39.83 deg; joints [46.494, -79.803, 89.678, -0.873, 80.104, 46.64]
  MoveL 221 to (130.96, 23.01, 0) mm, rotated rx 180 ry 0 rz -39.83 deg; joints [46.527, -79.75, 89.616, -0.873, 80.114, 46.674]
  MoveL 222 to (131.5, 23.71, 0) mm, rotated rx -180 ry 0 rz -39.83 deg; joints [46.559, -79.696, 89.553, -0.873, 80.123, 46.706]
  MoveL 223 to (132.03, 24.41, 0) mm, rotated rx 180 ry 0 rz -39.83 deg; joints [46.591, -79.641, 89.488, -0.873, 80.133, 46.737]
  MoveL 224 to (132.03, 24.41, 0) mm, rotated rx 180 ry 0 rz -39.83 deg; joints [46.591, -79.641, 89.488, -0.873, 80.133, 46.737]
  MoveL 225 to (133.61, 25.02, 0) mm, rotated rx 180 ry 0 rz -39.83 deg; joints [46.68, -79.599, 89.44, -0.873, 80.141, 46.826]
  MoveL 226 to (135.19, 25.64, 0) mm, rotated rx 180 ry 0 rz -39.83 deg; joints [46.769, -79.555, 89.39, -0.873, 80.148, 46.915]
  MoveL 227 to (136.75, 26.27, 0) mm, rotated rx 180 ry 0 rz -39.83 deg; joints [46.857, -79.51, 89.339, -0.873, 80.156, 47.003]
  MoveL 228 to (138.31, 26.93, 0) mm, rotated rx 180 ry 0 rz -39.83 deg; joints [46.945, -79.463, 89.284, -0.873, 80.164, 47.091]
  MoveL 229 to (139.71, 27.55, 0) mm, rotated rx 180 ry 0 rz -39.83 deg; joints [47.024, -79.418, 89.233, -0.873, 80.172, 47.17]
  MoveL 230 to (141.09, 28.2, 0) mm, rotated rx 180 ry 0 rz -39.83 deg; joints [47.102, -79.371, 89.178, -0.873, 80.18, 47.248]
  MoveL 231 to (142.46, 28.87, 0) mm, rotated rx -180 ry 0 rz -39.83 deg; joints [47.18, -79.321, 89.121, -0.873, 80.189, 47.325]
  MoveL 232 to (143.82, 29.58, 0) mm, rotated rx 180 ry 0 rz -39.83 deg; joints [47.256, -79.268, 89.06, -0.873, 80.199, 47.402]
  MoveL 233 to (144.91, 30.17, 0) mm, rotated rx 180 ry 0 rz -39.83 deg; joints [47.318, -79.224, 89.008, -0.873, 80.207, 47.463]
  MoveL 234 to (145.99, 30.78, 0) mm, rotated rx 180 ry 0 rz -39.83 deg; joints [47.379, -79.178, 88.955, -0.873, 80.215, 47.524]
  MoveL 235 to (147.07, 31.41, 0) mm, rotated rx 180 ry 0 rz -39.83 deg; joints [47.439, -79.13, 88.899, -0.873, 80.224, 47.584]
  MoveL 236 to (148.13, 32.05, 0) mm, rotated rx -180 ry 0 rz -39.83 deg; joints [47.5, -79.081, 88.842, -0.873, 80.233, 47.644]
  MoveL 237 to (148.99, 32.58, 0) mm, rotated rx 180 ry 0 rz -39.83 deg; joints [47.548, -79.041, 88.795, -0.873, 80.24, 47.693]
  MoveL 238 to (149.83, 33.11, 0) mm, rotated rx 180 ry 0 rz -39.83 deg; joints [47.596, -79, 88.747, -0.873, 80.248, 47.74]
  MoveL 239 to (150.67, 33.66, 0) mm, rotated rx -180 ry 0 rz -39.83 deg; joints [47.643, -78.958, 88.698, -0.873, 80.256, 47.788]
  MoveL 240 to (151.5, 34.23, 0) mm, rotated rx 180 ry 0 rz -39.83 deg; joints [47.69, -78.914, 88.647, -0.873, 80.264, 47.834]
  MoveL 241 to (152.71, 35.09, 0) mm, rotated rx 180 ry 0 rz -39.83 deg; joints [47.758, -78.847, 88.567, -0.873, 80.277, 47.902]
  MoveL 242 to (153.9, 35.99, 0) mm, rotated rx 180 ry 0 rz -39.83 deg; joints [47.825, -78.777, 88.485, -0.873, 80.291, 47.969]
  MoveL 243 to (155.07, 36.91, 0) mm, rotated rx 180 ry 0 rz -39.83 deg; joints [47.891, -78.705, 88.4, -0.873, 80.305, 48.035]
  MoveL 244 to (156.23, 37.83, 0) mm, rotated rx 180 ry 0 rz -39.83 deg; joints [47.956, -78.633, 88.314, -0.873, 80.319, 48.1]
  MoveL 245 to (156.23, 37.83, 0) mm, rotated rx 180 ry 0 rz -39.83 deg; joints [47.956, -78.633, 88.314, -0.873, 80.319, 48.1]
  MoveL 246 to (157.43, 38.33, 0) mm, rotated rx 180 ry 0 rz -39.83 deg; joints [48.023, -78.595, 88.271, -0.873, 80.326, 48.167]
  MoveL 247 to (158.63, 38.84, 0) mm, rotated rx 180 ry 0 rz -39.83 deg; joints [48.089, -78.557, 88.226, -0.873, 80.333, 48.232]
  MoveL 248 to (159.8, 39.38, 0) mm, rotated rx 180 ry 0 rz -39.83 deg; joints [48.154, -78.515, 88.178, -0.873, 80.341, 48.298]
  MoveL 249 to (160.96, 39.96, 0) mm, rotated rx 180 ry 0 rz -39.83 deg; joints [48.218, -78.471, 88.125, -0.873, 80.35, 48.362]
  MoveL 250 to (161.75, 40.4, 0) mm, rotated rx -180 ry 0 rz -39.83 deg; joints [48.262, -78.437, 88.085, -0.873, 80.357, 48.405]
  MoveL 251 to (162.53, 40.86, 0) mm, rotated rx 180 ry 0 rz -39.83 deg; joints [48.306, -78.4, 88.043, -0.873, 80.364, 48.449]
  MoveL 252 to (163.3, 41.34, 0) mm, rotated rx -180 ry 0 rz -39.83 deg; joints [48.348, -78.363, 87.998, -0.873, 80.371, 48.491]
  MoveL 253 to (164.06, 41.83, 0) mm, rotated rx 180 ry 0 rz -39.83 deg; joints [48.391, -78.324, 87.953, -0.873, 80.379, 48.534]
  MoveL 254 to (165.06, 42.49, 0) mm, rotated rx 180 ry 0 rz -39.83 deg; joints [48.446, -78.273, 87.891, -0.873, 80.389, 48.589]
  MoveL 255 to (166.04, 43.16, 0) mm, rotated rx 180 ry 0 rz -39.83 deg; joints [48.5, -78.219, 87.828, -0.873, 80.4, 48.643]
  MoveL 256 to (167, 43.86, 0) mm, rotated rx 180 ry 0 rz -39.83 deg; joints [48.554, -78.164, 87.762, -0.873, 80.411, 48.696]
  MoveL 257 to (167.94, 44.59, 0) mm, rotated rx 180 ry 0 rz -39.83 deg; joints [48.606, -78.105, 87.692, -0.873, 80.423, 48.748]
  MoveL 258 to (168.74, 45.27, 0) mm, rotated rx -180 ry 0 rz -39.83 deg; joints [48.65, -78.051, 87.628, -0.873, 80.435, 48.792]
  MoveL 259 to (169.52, 45.98, 0) mm, rotated rx 180 ry 0 rz -39.83 deg; joints [48.694, -77.994, 87.559, -0.873, 80.447, 48.835]
  MoveL 260 to (170.27, 46.72, 0) mm, rotated rx 180 ry 0 rz -39.83 deg; joints [48.736, -77.935, 87.488, -0.873, 80.459, 48.877]
  MoveL 261 to (171, 47.49, 0) mm, rotated rx -180 ry 0 rz -39.83 deg; joints [48.776, -77.873, 87.414, -0.873, 80.472, 48.917]
  MoveL 262 to (171.86, 48.46, 0) mm, rotated rx 180 ry 0 rz -39.83 deg; joints [48.824, -77.794, 87.32, -0.873, 80.489, 48.965]
  MoveL 263 to (172.69, 49.47, 0) mm, rotated rx -180 ry 0 rz -39.83 deg; joints [48.87, -77.713, 87.221, -0.872, 80.506, 49.011]
  MoveL 264 to (173.49, 50.49, 0) mm, rotated rx 180 ry 0 rz -39.83 deg; joints [48.915, -77.63, 87.121, -0.872, 80.524, 49.055]
  MoveL 265 to (174.28, 51.54, 0) mm, rotated rx 180 ry 0 rz -39.83 deg; joints [48.958, -77.545, 87.019, -0.872, 80.543, 49.098]
  MoveL 266 to (175, 52.51, 0) mm, rotated rx -180 ry 0 rz -39.83 deg; joints [48.998, -77.466, 86.923, -0.872, 80.56, 49.138]
  MoveL 267 to (175.7, 53.5, 0) mm, rotated rx 180 ry 0 rz -39.83 deg; joints [49.037, -77.386, 86.825, -0.872, 80.578, 49.177]
  MoveL 268 to (176.38, 54.5, 0) mm, rotated rx 180 ry 0 rz -39.83 deg; joints [49.074, -77.304, 86.726, -0.872, 80.596, 49.214]
  MoveL 269 to (177, 55.53, 0) mm, rotated rx 180 ry 0 rz -39.83 deg; joints [49.109, -77.22, 86.624, -0.872, 80.615, 49.248]
  MoveL 270 to (177.65, 56.72, 0) mm, rotated rx -180 ry 0 rz -39.83 deg; joints [49.145, -77.123, 86.505, -0.872, 80.637, 49.284]
  MoveL 271 to (178.22, 57.94, 0) mm, rotated rx -180 ry 0 rz -39.83 deg; joints [49.177, -77.023, 86.383, -0.872, 80.66, 49.315]
  MoveL 272 to (178.75, 59.19, 0) mm, rotated rx 180 ry 0 rz -39.83 deg; joints [49.206, -76.921, 86.257, -0.872, 80.683, 49.344]
  MoveL 273 to (179.22, 60.46, 0) mm, rotated rx 180 ry 0 rz -39.83 deg; joints [49.232, -76.817, 86.129, -0.872, 80.707, 49.37]
  MoveL 274 to (180.02, 63, 0) mm, rotated rx 180 ry 0 rz -39.83 deg; joints [49.278, -76.609, 85.873, -0.872, 80.757, 49.415]
  MoveL 275 to (180.7, 65.58, 0) mm, rotated rx -180 ry 0 rz -39.83 deg; joints [49.316, -76.397, 85.611, -0.872, 80.807, 49.452]
  MoveL 276 to (181.29, 68.18, 0) mm, rotated rx -180 ry 0 rz -39.83 deg; joints [49.349, -76.184, 85.346, -0.871, 80.859, 49.485]
  MoveL 277 to (181.83, 70.79, 0) mm, rotated rx 180 ry 0 rz -39.83 deg; joints [49.38, -75.969, 85.079, -0.871, 80.913, 49.515]
  MoveL 278 to (181.83, 70.79, 0) mm, rotated rx 180 ry 0 rz -39.83 deg; joints [49.38, -75.969, 85.079, -0.871, 80.913, 49.515]
  MoveL 279 to (182.64, 72.73, 0) mm, rotated rx 180 ry 0 rz -39.83 deg; joints [49.424, -75.81, 84.88, -0.871, 80.952, 49.558]
  MoveL 280 to (183.42, 74.68, 0) mm, rotated rx 180 ry 0 rz -39.83 deg; joints [49.467, -75.649, 84.68, -0.871, 80.993, 49.6]
  MoveL 281 to (184.16, 76.65, 0) mm, rotated rx 180 ry 0 rz -39.83 deg; joints [49.507, -75.488, 84.478, -0.871, 81.034, 49.64]
  MoveL 282 to (184.84, 78.63, 0) mm, rotated rx -180 ry 0 rz -39.83 deg; joints [49.544, -75.325, 84.273, -0.871, 81.076, 49.676]
  MoveL 283 to (185.49, 80.78, 0) mm, rotated rx -180 ry 0 rz -39.83 deg; joints [49.579, -75.147, 84.049, -0.871, 81.123, 49.711]
  MoveL 284 to (186.06, 82.96, 0) mm, rotated rx 180 ry 0 rz -39.83 deg; joints [49.611, -74.968, 83.823, -0.871, 81.17, 49.741]
  MoveL 285 to (186.59, 85.15, 0) mm, rotated rx 180 ry 0 rz -39.83 deg; joints [49.639, -74.787, 83.594, -0.87, 81.219, 49.769]
  MoveL 286 to (187.09, 87.35, 0) mm, rotated rx -180 ry 0 rz -39.83 deg; joints [49.667, -74.605, 83.363, -0.87, 81.268, 49.796]
  MoveL 287 to (187.09, 87.35, 0) mm, rotated rx -180 ry 0 rz -39.83 deg; joints [49.667, -74.605, 83.363, -0.87, 81.268, 49.796]
  MoveL 288 to (187.84, 88.11, 0) mm, rotated rx 180 ry 0 rz -39.83 deg; joints [49.706, -74.543, 83.285, -0.87, 81.285, 49.835]
  MoveL 289 to (188.58, 88.88, 0) mm, rotated rx 180 ry 0 rz -39.83 deg; joints [49.745, -74.479, 83.205, -0.87, 81.302, 49.874]
  MoveL 290 to (189.29, 89.67, 0) mm, rotated rx 180 ry 0 rz -39.83 deg; joints [49.782, -74.414, 83.123, -0.87, 81.319, 49.911]
  MoveL 291 to (189.97, 90.49, 0) mm, rotated rx 180 ry 0 rz -39.83 deg; joints [49.818, -74.347, 83.038, -0.87, 81.338, 49.946]
  MoveL 292 to (190.77, 91.59, 0) mm, rotated rx 180 ry 0 rz -39.83 deg; joints [49.86, -74.256, 82.923, -0.87, 81.363, 49.987]
  MoveL 293 to (191.49, 92.73, 0) mm, rotated rx 180 ry 0 rz -39.83 deg; joints [49.898, -74.162, 82.803, -0.87, 81.389, 50.025]
  MoveL 294 to (192.16, 93.91, 0) mm, rotated rx -180 ry 0 rz -39.83 deg; joints [49.933, -74.064, 82.678, -0.87, 81.416, 50.06]
  MoveL 295 to (192.79, 95.12, 0) mm, rotated rx 180 ry 0 rz -39.83 deg; joints [49.966, -73.964, 82.55, -0.87, 81.444, 50.092]
  MoveL 296 to (193.42, 96.41, 0) mm, rotated rx -180 ry 0 rz -39.83 deg; joints [49.998, -73.858, 82.415, -0.87, 81.474, 50.124]
  MoveL 297 to (194, 97.71, 0) mm, rotated rx 180 ry 0 rz -39.83 deg; joints [50.029, -73.75, 82.277, -0.87, 81.505, 50.154]
  MoveL 298 to (194.54, 99.02, 0) mm, rotated rx 180 ry 0 rz -39.83 deg; joints [50.057, -73.641, 82.137, -0.87, 81.536, 50.182]
  MoveL 299 to (195.01, 100.36, 0) mm, rotated rx 180 ry 0 rz -39.83 deg; joints [50.081, -73.53, 81.994, -0.869, 81.569, 50.206]
  MoveL 300 to (195.32, 101.38, 0) mm, rotated rx 180 ry 0 rz -39.83 deg; joints [50.097, -73.446, 81.885, -0.869, 81.593, 50.222]
  MoveL 301 to (195.6, 102.4, 0) mm, rotated rx -180 ry 0 rz -39.83 deg; joints [50.112, -73.361, 81.776, -0.869, 81.618, 50.236]
  MoveL 302 to (195.86, 103.44, 0) mm, rotated rx 180 ry 0 rz -39.83 deg; joints [50.125, -73.275, 81.665, -0.869, 81.643, 50.248]
  MoveL 303 to (196.09, 104.48, 0) mm, rotated rx 180 ry 0 rz -39.83 deg; joints [50.137, -73.188, 81.553, -0.869, 81.669, 50.26]
  MoveL 304 to (196.37, 105.93, 0) mm, rotated rx 180 ry 0 rz -39.83 deg; joints [50.151, -73.068, 81.396, -0.869, 81.705, 50.274]
  MoveL 305 to (196.61, 107.39, 0) mm, rotated rx 180 ry 0 rz -39.83 deg; joints [50.164, -72.947, 81.239, -0.869, 81.741, 50.285]
  MoveL 306 to (196.78, 108.85, 0) mm, rotated rx -180 ry 0 rz -39.83 deg; joints [50.173, -72.825, 81.081, -0.869, 81.778, 50.294]
  MoveL 307 to (196.89, 110.32, 0) mm, rotated rx 180 ry 0 rz -39.83 deg; joints [50.178, -72.703, 80.922, -0.869, 81.815, 50.299]
  MoveL 308 to (196.92, 111.83, 0) mm, rotated rx -180 ry 0 rz -39.83 deg; joints [50.18, -72.577, 80.757, -0.869, 81.854, 50.3]
  MoveL 309 to (196.88, 113.35, 0) mm, rotated rx -180 ry 0 rz -39.83 deg; joints [50.178, -72.451, 80.592, -0.869, 81.893, 50.297]
  MoveL 310 to (196.78, 114.86, 0) mm, rotated rx 180 ry 0 rz -39.83 deg; joints [50.172, -72.325, 80.426, -0.869, 81.932, 50.291]
  MoveL 311 to (196.62, 116.38, 0) mm, rotated rx 180 ry 0 rz -39.83 deg; joints [50.164, -72.199, 80.26, -0.869, 81.972, 50.283]
  MoveL 312 to (196.41, 117.98, 0) mm, rotated rx 180 ry 0 rz -39.83 deg; joints [50.154, -72.066, 80.085, -0.868, 82.014, 50.272]
  MoveL 313 to (196.15, 119.56, 0) mm, rotated rx -180 ry 0 rz -39.83 deg; joints [50.141, -71.933, 79.91, -0.868, 82.057, 50.258]
  MoveL 314 to (195.82, 121.14, 0) mm, rotated rx -180 ry 0 rz -39.83 deg; joints [50.124, -71.802, 79.737, -0.868, 82.099, 50.24]
  MoveL 315 to (195.41, 122.69, 0) mm, rotated rx 180 ry 0 rz -39.83 deg; joints [50.103, -71.673, 79.565, -0.868, 82.141, 50.219]
  MoveL 316 to (194.83, 124.46, 0) mm, rotated rx -180 ry 0 rz -39.83 deg; joints [50.074, -71.525, 79.369, -0.868, 82.189, 50.189]
  MoveL 317 to (194.14, 126.19, 0) mm, rotated rx -180 ry 0 rz -39.83 deg; joints [50.04, -71.381, 79.176, -0.868, 82.237, 50.154]
  MoveL 318 to (193.37, 127.88, 0) mm, rotated rx 180 ry 0 rz -39.83 deg; joints [50.001, -71.239, 78.986, -0.868, 82.284, 50.114]
  MoveL 319 to (192.52, 129.55, 0) mm, rotated rx 180 ry 0 rz -39.83 deg; joints [49.958, -71.1, 78.8, -0.868, 82.331, 50.071]
  MoveL 320 to (191.8, 130.85, 0) mm, rotated rx -180 ry 0 rz -39.83 deg; joints [49.922, -70.991, 78.653, -0.868, 82.368, 50.035]
  MoveL 321 to (191.04, 132.13, 0) mm, rotated rx 180 ry 0 rz -39.83 deg; joints [49.884, -70.884, 78.509, -0.868, 82.404, 49.996]
  MoveL 322 to (190.23, 133.37, 0) mm, rotated rx 180 ry 0 rz -39.83 deg; joints [49.844, -70.779, 78.368, -0.868, 82.44, 49.955]
  MoveL 323 to (189.36, 134.58, 0) mm, rotated rx 180 ry 0 rz -39.83 deg; joints [49.801, -70.677, 78.231, -0.868, 82.475, 49.912]
  MoveL 324 to (188.26, 135.97, 0) mm, rotated rx 180 ry 0 rz -39.83 deg; joints [49.746, -70.561, 78.074, -0.868, 82.515, 49.856]
  MoveL 325 to (187.07, 137.28, 0) mm, rotated rx -180 ry 0 rz -39.83 deg; joints [49.688, -70.451, 77.923, -0.868, 82.554, 49.797]
  MoveL 326 to (185.8, 138.51, 0) mm, rotated rx 180 ry 0 rz -39.83 deg; joints [49.625, -70.347, 77.782, -0.868, 82.59, 49.734]
  MoveL 327 to (184.45, 139.64, 0) mm, rotated rx 180 ry 0 rz -39.83 deg; joints [49.558, -70.25, 77.651, -0.867, 82.624, 49.666]
  MoveL 328 to (183.43, 140.4, 0) mm, rotated rx -180 ry 0 rz -39.83 deg; joints [49.508, -70.186, 77.562, -0.867, 82.648, 49.616]
  MoveL 329 to (182.37, 141.12, 0) mm, rotated rx -180 ry 0 rz -39.83 deg; joints [49.456, -70.125, 77.478, -0.867, 82.669, 49.563]
  MoveL 330 to (181.3, 141.81, 0) mm, rotated rx 180 ry 0 rz -39.83 deg; joints [49.403, -70.066, 77.398, -0.867, 82.691, 49.51]
  MoveL 331 to (180.22, 142.49, 0) mm, rotated rx -180 ry 0 rz -39.83 deg; joints [49.349, -70.008, 77.318, -0.867, 82.712, 49.456]
  MoveL 332 to (180.22, 142.49, 0) mm, rotated rx -180 ry 0 rz -39.83 deg; joints [49.349, -70.008, 77.318, -0.867, 82.712, 49.456]
  MoveL 333 to (180.07, 143, 0) mm, rotated rx 180 ry 0 rz -39.83 deg; joints [49.342, -69.965, 77.259, -0.867, 82.727, 49.449]
  MoveL 334 to (179.92, 143.51, 0) mm, rotated rx 180 ry 0 rz -39.83 deg; joints [49.335, -69.921, 77.2, -0.867, 82.742, 49.442]
  MoveL 335 to (179.75, 144.02, 0) mm, rotated rx -180 ry 0 rz -39.83 deg; joints [49.327, -69.879, 77.142, -0.867, 82.758, 49.434]
  MoveL 336 to (179.56, 144.52, 0) mm, rotated rx -180 ry 0 rz -39.83 deg; joints [49.318, -69.837, 77.085, -0.867, 82.773, 49.424]
  MoveL 337 to (179.38, 144.94, 0) mm, rotated rx 180 ry 0 rz -39.83 deg; joints [49.309, -69.801, 77.037, -0.867, 82.785, 49.415]
  MoveL 338 to (179.17, 145.35, 0) mm, rotated rx 180 ry 0 rz -39.83 deg; joints [49.3, -69.766, 76.989, -0.867, 82.798, 49.405]
  MoveL 339 to (178.96, 145.76, 0) mm, rotated rx -180 ry 0 rz -39.83 deg; joints [49.289, -69.731, 76.942, -0.867, 82.81, 49.395]
  MoveL 340 to (178.74, 146.17, 0) mm, rotated rx 180 ry 0 rz -39.83 deg; joints [49.279, -69.697, 76.894, -0.867, 82.823, 49.384]
  MoveL 341 to (178.74, 146.17, 0) mm, rotated rx 180 ry 0 rz -39.83 deg; joints [49.279, -69.697, 76.894, -0.867, 82.823, 49.384]
  MoveL 342 to (178.76, 147.55, 0) mm, rotated rx 180 ry 0 rz -39.83 deg; joints [49.281, -69.58, 76.736, -0.867, 82.865, 49.385]
  MoveL 343 to (178.76, 148.94, 0) mm, rotated rx -180 ry 0 rz -39.83 deg; joints [49.282, -69.463, 76.576, -0.867, 82.907, 49.386]
  MoveL 344 to (178.74, 150.33, 0) mm, rotated rx 180 ry 0 rz -39.83 deg; joints [49.282, -69.346, 76.417, -0.867, 82.949, 49.385]
  MoveL 345 to (178.69, 151.72, 0) mm, rotated rx -180 ry 0 rz -39.83 deg; joints [49.281, -69.228, 76.257, -0.867, 82.992, 49.383]
  MoveL 346 to (178.61, 152.98, 0) mm, rotated rx 180 ry 0 rz -39.83 deg; joints [49.278, -69.121, 76.111, -0.867, 83.031, 49.38]
  MoveL 347 to (178.49, 154.25, 0) mm, rotated rx 180 ry 0 rz -39.83 deg; joints [49.273, -69.014, 75.965, -0.867, 83.07, 49.374]
  MoveL 348 to (178.33, 155.51, 0) mm, rotated rx 180 ry 0 rz -39.83 deg; joints [49.266, -68.908, 75.818, -0.867, 83.11, 49.367]
  MoveL 349 to (178.11, 156.76, 0) mm, rotated rx 180 ry 0 rz -39.83 deg; joints [49.256, -68.802, 75.673, -0.867, 83.149, 49.356]
  MoveL 350 to (177.84, 158.04, 0) mm, rotated rx 180 ry 0 rz -39.83 deg; joints [49.244, -68.693, 75.523, -0.867, 83.19, 49.343]
  MoveL 351 to (177.51, 159.31, 0) mm, rotated rx -180 ry 0 rz -39.83 deg; joints [49.229, -68.585, 75.374, -0.866, 83.23, 49.328]
  MoveL 352 to (177.13, 160.56, 0) mm, rotated rx -180 ry 0 rz -39.83 deg; joints [49.211, -68.478, 75.227, -0.866, 83.271, 49.31]
  MoveL 353 to (176.7, 161.8, 0) mm, rotated rx 180 ry 0 rz -39.83 deg; joints [49.191, -68.373, 75.081, -0.866, 83.311, 49.289]
  MoveL 354 to (176.08, 163.33, 0) mm, rotated rx 180 ry 0 rz -39.83 deg; joints [49.162, -68.242, 74.9, -0.866, 83.361, 49.259]
  MoveL 355 to (175.39, 164.83, 0) mm, rotated rx -180 ry 0 rz -39.83 deg; joints [49.13, -68.113, 74.721, -0.866, 83.41, 49.226]
  MoveL 356 to (174.65, 166.31, 0) mm, rotated rx 180 ry 0 rz -39.83 deg; joints [49.095, -67.986, 74.544, -0.866, 83.459, 49.19]
  MoveL 357 to (173.87, 167.78, 0) mm, rotated rx 180 ry 0 rz -39.83 deg; joints [49.058, -67.861, 74.369, -0.866, 83.508, 49.153]
  MoveL 358 to (173.21, 168.94, 0) mm, rotated rx -180 ry 0 rz -39.83 deg; joints [49.028, -67.76, 74.229, -0.866, 83.548, 49.122]
  MoveL 359 to (172.53, 170.09, 0) mm, rotated rx -180 ry 0 rz -39.83 deg; joints [48.996, -67.661, 74.091, -0.866, 83.586, 49.089]
  MoveL 360 to (171.81, 171.21, 0) mm, rotated rx 180 ry 0 rz -39.83 deg; joints [48.962, -67.565, 73.956, -0.866, 83.624, 49.055]
  MoveL 361 to (171.03, 172.28, 0) mm, rotated rx 180 ry 0 rz -39.83 deg; joints [48.925, -67.472, 73.826, -0.866, 83.661, 49.018]
  MoveL 362 to (170.01, 173.51, 0) mm, rotated rx 180 ry 0 rz -39.83 deg; joints [48.877, -67.366, 73.676, -0.866, 83.704, 48.969]
  MoveL 363 to (168.92, 174.67, 0) mm, rotated rx 180 ry 0 rz -39.83 deg; joints [48.825, -67.265, 73.534, -0.866, 83.744, 48.917]
  MoveL 364 to (167.76, 175.78, 0) mm, rotated rx 180 ry 0 rz -39.83 deg; joints [48.771, -67.168, 73.397, -0.866, 83.784, 48.861]
  MoveL 365 to (166.56, 176.85, 0) mm, rotated rx 180 ry 0 rz -39.83 deg; joints [48.714, -67.073, 73.263, -0.866, 83.822, 48.804]
  MoveL 366 to (165.14, 178.06, 0) mm, rotated rx 180 ry 0 rz -39.83 deg; joints [48.647, -66.967, 73.112, -0.866, 83.865, 48.737]
  MoveL 367 to (163.69, 179.21, 0) mm, rotated rx 180 ry 0 rz -39.83 deg; joints [48.579, -66.865, 72.967, -0.865, 83.907, 48.668]
  MoveL 368 to (162.18, 180.29, 0) mm, rotated rx 180 ry 0 rz -39.83 deg; joints [48.508, -66.769, 72.831, -0.865, 83.947, 48.596]
  MoveL 369 to (160.62, 181.27, 0) mm, rotated rx 180 ry 0 rz -39.83 deg; joints [48.434, -66.681, 72.705, -0.865, 83.983, 48.522]
  MoveL 370 to (159.66, 181.8, 0) mm, rotated rx 180 ry 0 rz -39.83 deg; joints [48.389, -66.634, 72.638, -0.865, 84.003, 48.476]
  MoveL 371 to (158.68, 182.29, 0) mm, rotated rx 180 ry 0 rz -39.83 deg; joints [48.342, -66.589, 72.574, -0.865, 84.022, 48.429]
  MoveL 372 to (157.68, 182.76, 0) mm, rotated rx 180 ry 0 rz -39.83 deg; joints [48.295, -66.546, 72.512, -0.865, 84.04, 48.382]
  MoveL 373 to (156.68, 183.22, 0) mm, rotated rx 180 ry 0 rz -39.83 deg; joints [48.248, -66.504, 72.451, -0.865, 84.058, 48.335]
  MoveL 374 to (156.68, 183.22, 0) mm, rotated rx 180 ry 0 rz -39.83 deg; joints [48.248, -66.504, 72.451, -0.865, 84.058, 48.335]
  MoveL 375 to (156.82, 183.34, 0) mm, rotated rx 180 ry 0 rz -39.83 deg; joints [48.255, -66.494, 72.437, -0.865, 84.062, 48.341]
  MoveL 376 to (156.96, 183.47, 0) mm, rotated rx 180 ry 0 rz -39.83 deg; joints [48.262, -66.484, 72.422, -0.865, 84.066, 48.348]
  MoveL 377 to (157.11, 183.58, 0) mm, rotated rx 180 ry 0 rz -39.83 deg; joints [48.269, -66.474, 72.409, -0.865, 84.07, 48.356]
  MoveL 378 to (157.26, 183.68, 0) mm, rotated rx 180 ry 0 rz -39.83 deg; joints [48.277, -66.466, 72.398, -0.865, 84.073, 48.363]
  MoveL 379 to (157.57, 183.82, 0) mm, rotated rx -180 ry 0 rz -39.83 deg; joints [48.292, -66.455, 72.383, -0.865, 84.077, 48.378]
  MoveL 380 to (157.9, 183.91, 0) mm, rotated rx -180 ry 0 rz -39.83 deg; joints [48.308, -66.448, 72.373, -0.865, 84.08, 48.394]
  MoveL 381 to (158.24, 183.98, 0) mm, rotated rx 180 ry 0 rz -39.83 deg; joints [48.324, -66.442, 72.366, -0.865, 84.082, 48.41]
  MoveL 382 to (158.58, 184.05, 0) mm, rotated rx 180 ry 0 rz -39.83 deg; joints [48.341, -66.438, 72.36, -0.865, 84.084, 48.427]
  MoveL 383 to (159.29, 184.23, 0) mm, rotated rx 180 ry 0 rz -39.83 deg; joints [48.375, -66.424, 72.342, -0.865, 84.089, 48.461]
  MoveL 384 to (159.97, 184.45, 0) mm, rotated rx -180 ry 0 rz -39.83 deg; joints [48.408, -66.406, 72.317, -0.865, 84.096, 48.494]
  MoveL 385 to (160.64, 184.71, 0) mm, rotated rx 180 ry 0 rz -39.83 deg; joints [48.44, -66.386, 72.29, -0.865, 84.104, 48.526]
  MoveL 386 to (161.32, 184.97, 0) mm, rotated rx 180 ry 0 rz -39.83 deg; joints [48.473, -66.365, 72.261, -0.865, 84.112, 48.559]
  MoveL 387 to (161.8, 185.16, 0) mm, rotated rx 180 ry 0 rz -39.83 deg; joints [48.496, -66.35, 72.241, -0.865, 84.118, 48.582]
  MoveL 388 to (162.28, 185.35, 0) mm, rotated rx 180 ry 0 rz -39.83 deg; joints [48.52, -66.335, 72.22, -0.865, 84.124, 48.605]
  MoveL 389 to (162.75, 185.57, 0) mm, rotated rx 180 ry 0 rz -39.83 deg; joints [48.542, -66.317, 72.195, -0.865, 84.131, 48.628]
  MoveL 390 to (163.18, 185.83, 0) mm, rotated rx 180 ry 0 rz -39.83 deg; joints [48.564, -66.295, 72.165, -0.865, 84.14, 48.649]
  MoveL 391 to (163.55, 186.12, 0) mm, rotated rx 180 ry 0 rz -39.83 deg; joints [48.582, -66.271, 72.131, -0.865, 84.149, 48.667]
  MoveL 392 to (163.89, 186.45, 0) mm, rotated rx 180 ry 0 rz -39.83 deg; joints [48.598, -66.243, 72.093, -0.865, 84.161, 48.683]
  MoveL 393 to (164.2, 186.81, 0) mm, rotated rx -180 ry 0 rz -39.83 deg; joints [48.613, -66.213, 72.05, -0.865, 84.173, 48.698]
  MoveL 394 to (164.48, 187.19, 0) mm, rotated rx 180 ry 0 rz -39.83 deg; joints [48.627, -66.181, 72.005, -0.865, 84.186, 48.712]
  MoveL 395 to (164.68, 187.5, 0) mm, rotated rx 180 ry 0 rz -39.83 deg; joints [48.637, -66.155, 71.969, -0.865, 84.197, 48.721]
  MoveL 396 to (164.86, 187.81, 0) mm, rotated rx 180 ry 0 rz -39.83 deg; joints [48.646, -66.128, 71.931, -0.865, 84.208, 48.73]
  MoveL 397 to (165.02, 188.14, 0) mm, rotated rx 180 ry 0 rz -39.83 deg; joints [48.654, -66.101, 71.892, -0.865, 84.219, 48.738]
  MoveL 398 to (165.16, 188.47, 0) mm, rotated rx 180 ry 0 rz -39.83 deg; joints [48.662, -66.072, 71.852, -0.865, 84.231, 48.746]
  MoveL 399 to (165.23, 188.65, 0) mm, rotated rx 180 ry 0 rz -39.83 deg; joints [48.665, -66.057, 71.831, -0.865, 84.237, 48.749]
  MoveL 400 to (165.28, 188.82, 0) mm, rotated rx 180 ry 0 rz -39.83 deg; joints [48.668, -66.042, 71.809, -0.865, 84.243, 48.751]
  MoveL 401 to (165.32, 189, 0) mm, rotated rx 180 ry 0 rz -39.83 deg; joints [48.67, -66.026, 71.788, -0.865, 84.25, 48.754]
  MoveL 402 to (165.35, 189.18, 0) mm, rotated rx 180 ry 0 rz -39.83 deg; joints [48.671, -66.011, 71.766, -0.865, 84.256, 48.755]
  MoveL 403 to (165.36, 189.35, 0) mm, rotated rx 180 ry 0 rz -39.83 deg; joints [48.672, -65.996, 71.745, -0.865, 84.262, 48.755]
  MoveL 404 to (165.35, 189.53, 0) mm, rotated rx -180 ry 0 rz -39.83 deg; joints [48.672, -65.981, 71.724, -0.865, 84.269, 48.755]
  MoveL 405 to (165.33, 189.7, 0) mm, rotated rx 180 ry 0 rz -39.83 deg; joints [48.671, -65.966, 71.703, -0.865, 84.275, 48.754]
  MoveL 406 to (165.31, 189.87, 0) mm, rotated rx 180 ry 0 rz -39.83 deg; joints [48.67, -65.952, 71.682, -0.865, 84.281, 48.753]
  MoveL 407 to (165.31, 189.87, 0) mm, rotated rx 180 ry 0 rz -39.83 deg; joints [48.67, -65.952, 71.682, -0.865, 84.281, 48.753]
  MoveL 408 to (166.15, 190.18, 0) mm, rotated rx 180 ry 0 rz -39.83 deg; joints [48.711, -65.926, 71.647, -0.865, 84.291, 48.794]
  MoveL 409 to (166.99, 190.51, 0) mm, rotated rx 180 ry 0 rz -39.83 deg; joints [48.751, -65.9, 71.611, -0.865, 84.302, 48.834]
  MoveL 410 to (167.81, 190.85, 0) mm, rotated rx 180 ry 0 rz -39.83 deg; joints [48.791, -65.872, 71.571, -0.865, 84.313, 48.874]
  MoveL 411 to (168.62, 191.24, 0) mm, rotated rx 180 ry 0 rz -39.83 deg; joints [48.83, -65.84, 71.528, -0.865, 84.326, 48.912]
  MoveL 412 to (169.24, 191.57, 0) mm, rotated rx 180 ry 0 rz -39.83 deg; joints [48.86, -65.812, 71.489, -0.865, 84.337, 48.942]
  MoveL 413 to (169.84, 191.94, 0) mm, rotated rx 180 ry 0 rz -39.83 deg; joints [48.889, -65.781, 71.446, -0.865, 84.35, 48.971]
  MoveL 414 to (170.42, 192.34, 0) mm, rotated rx 180 ry 0 rz -39.83 deg; joints [48.917, -65.748, 71.399, -0.865, 84.363, 48.999]
  MoveL 415 to (170.97, 192.78, 0) mm, rotated rx -180 ry 0 rz -39.83 deg; joints [48.944, -65.71, 71.347, -0.865, 84.379, 49.025]
  MoveL 416 to (171.39, 193.17, 0) mm, rotated rx 180 ry 0 rz -39.83 deg; joints [48.964, -65.678, 71.301, -0.865, 84.392, 49.045]
  MoveL 417 to (171.78, 193.58, 0) mm, rotated rx 180 ry 0 rz -39.83 deg; joints [48.983, -65.643, 71.251, -0.865, 84.407, 49.064]
  MoveL 418 to (172.14, 194.03, 0) mm, rotated rx -180 ry 0 rz -39.83 deg; joints [49, -65.605, 71.198, -0.865, 84.423, 49.081]
  MoveL 419 to (172.44, 194.5, 0) mm, rotated rx -180 ry 0 rz -39.83 deg; joints [49.015, -65.564, 71.14, -0.865, 84.44, 49.096]
  MoveL 420 to (172.6, 194.81, 0) mm, rotated rx 180 ry 0 rz -39.83 deg; joints [49.023, -65.537, 71.103, -0.865, 84.451, 49.103]
  MoveL 421 to (172.73, 195.13, 0) mm, rotated rx 180 ry 0 rz -39.83 deg; joints [49.03, -65.51, 71.064, -0.865, 84.463, 49.11]
  MoveL 422 to (172.85, 195.46, 0) mm, rotated rx 180 ry 0 rz -39.83 deg; joints [49.036, -65.482, 71.024, -0.865, 84.474, 49.116]
  MoveL 423 to (172.95, 195.79, 0) mm, rotated rx 180 ry 0 rz -39.83 deg; joints [49.04, -65.453, 70.983, -0.864, 84.487, 49.12]
  MoveL 424 to (173.04, 196.19, 0) mm, rotated rx -180 ry 0 rz -39.83 deg; joints [49.045, -65.418, 70.934, -0.864, 84.501, 49.125]
  MoveL 425 to (173.1, 196.59, 0) mm, rotated rx 180 ry 0 rz -39.83 deg; joints [49.049, -65.384, 70.884, -0.864, 84.516, 49.128]
  MoveL 426 to (173.16, 197, 0) mm, rotated rx 180 ry 0 rz -39.83 deg; joints [49.052, -65.349, 70.834, -0.864, 84.531, 49.131]
  MoveL 427 to (173.2, 197.4, 0) mm, rotated rx 180 ry 0 rz -39.83 deg; joints [49.054, -65.314, 70.784, -0.864, 84.546, 49.133]
  MoveL 428 to (173.2, 197.4, 0) mm, rotated rx 180 ry 0 rz -39.83 deg; joints [49.054, -65.314, 70.784, -0.864, 84.546, 49.133]
  MoveL 429 to (173.89, 197.88, 0) mm, rotated rx 180 ry 0 rz -39.83 deg; joints [49.087, -65.273, 70.727, -0.864, 84.563, 49.166]
  MoveL 430 to (174.56, 198.37, 0) mm, rotated rx -180 ry 0 rz -39.83 deg; joints [49.12, -65.232, 70.669, -0.864, 84.58, 49.198]
  MoveL 431 to (175.23, 198.87, 0) mm, rotated rx 180 ry 0 rz -39.83 deg; joints [49.152, -65.189, 70.61, -0.864, 84.598, 49.23]
  MoveL 432 to (175.88, 199.38, 0) mm, rotated rx 180 ry 0 rz -39.83 deg; joints [49.183, -65.145, 70.548, -0.864, 84.616, 49.261]
  MoveL 433 to (176.34, 199.76, 0) mm, rotated rx 180 ry 0 rz -39.83 deg; joints [49.205, -65.113, 70.502, -0.864, 84.63, 49.282]
  MoveL 434 to (176.78, 200.15, 0) mm, rotated rx 180 ry 0 rz -39.83 deg; joints [49.226, -65.08, 70.455, -0.864, 84.644, 49.303]
  MoveL 435 to (177.21, 200.55, 0) mm, rotated rx -180 ry 0 rz -39.83 deg; joints [49.247, -65.046, 70.407, -0.864, 84.659, 49.324]
  MoveL 436 to (177.65, 200.95, 0) mm, rotated rx -180 ry 0 rz -39.83 deg; joints [49.268, -65.011, 70.358, -0.864, 84.673, 49.345]
  MoveL 437 to (178.02, 201.32, 0) mm, rotated rx 180 ry 0 rz -39.83 deg; joints [49.286, -64.98, 70.313, -0.864, 84.687, 49.363]
  MoveL 438 to (178.38, 201.7, 0) mm, rotated rx -180 ry 0 rz -39.83 deg; joints [49.303, -64.947, 70.267, -0.864, 84.7, 49.38]
  MoveL 439 to (178.71, 202.1, 0) mm, rotated rx -180 ry 0 rz -39.83 deg; joints [49.319, -64.913, 70.218, -0.864, 84.715, 49.395]
  MoveL 440 to (178.99, 202.53, 0) mm, rotated rx 180 ry 0 rz -39.83 deg; joints [49.332, -64.876, 70.165, -0.864, 84.731, 49.408]
  MoveL 441 to (179.14, 202.84, 0) mm, rotated rx 180 ry 0 rz -39.83 deg; joints [49.34, -64.848, 70.126, -0.864, 84.743, 49.416]
  MoveL 442 to (179.28, 203.17, 0) mm, rotated rx 180 ry 0 rz -39.83 deg; joints [49.346, -64.82, 70.085, -0.864, 84.755, 49.422]
  MoveL 443 to (179.39, 203.51, 0) mm, rotated rx 180 ry 0 rz -39.83 deg; joints [49.352, -64.79, 70.043, -0.864, 84.768, 49.427]
  MoveL 444 to (179.48, 203.86, 0) mm, rotated rx 180 ry 0 rz -39.83 deg; joints [49.356, -64.76, 70, -0.864, 84.781, 49.432]
  MoveL 445 to (179.54, 204.16, 0) mm, rotated rx -180 ry 0 rz -39.83 deg; joints [49.359, -64.734, 69.963, -0.864, 84.793, 49.435]
  MoveL 446 to (179.59, 204.46, 0) mm, rotated rx 180 ry 0 rz -39.83 deg; joints [49.362, -64.708, 69.926, -0.864, 84.804, 49.437]
  MoveL 447 to (179.63, 204.75, 0) mm, rotated rx -180 ry 0 rz -39.83 deg; joints [49.364, -64.682, 69.888, -0.864, 84.815, 49.439]
  MoveL 448 to (179.65, 205.05, 0) mm, rotated rx 180 ry 0 rz -39.83 deg; joints [49.365, -64.656, 69.851, -0.864, 84.827, 49.44]
  MoveL 449 to (179.64, 205.4, 0) mm, rotated rx 180 ry 0 rz -39.83 deg; joints [49.365, -64.626, 69.808, -0.864, 84.84, 49.44]
  MoveL 450 to (179.62, 205.74, 0) mm, rotated rx 180 ry 0 rz -39.83 deg; joints [49.364, -64.596, 69.764, -0.864, 84.853, 49.439]
  MoveL 451 to (179.58, 206.09, 0) mm, rotated rx -180 ry 0 rz -39.83 deg; joints [49.363, -64.566, 69.721, -0.864, 84.866, 49.437]
  MoveL 452 to (179.54, 206.43, 0) mm, rotated rx 180 ry 0 rz -39.83 deg; joints [49.361, -64.536, 69.677, -0.864, 84.88, 49.435]
  MoveL 453 to (179.54, 206.43, 0) mm, rotated rx 180 ry 0 rz -39.83 deg; joints [49.361, -64.536, 69.677, -0.864, 84.88, 49.435]
  MoveL 454 to (180.03, 206.86, 0) mm, rotated rx 180 ry 0 rz -39.83 deg; joints [49.384, -64.499, 69.625, -0.864, 84.895, 49.458]
  MoveL 455 to (180.51, 207.29, 0) mm, rotated rx 180 ry 0 rz -39.83 deg; joints [49.407, -64.461, 69.572, -0.864, 84.912, 49.48]
  MoveL 456 to (180.97, 207.74, 0) mm, rotated rx -180 ry 0 rz -39.83 deg; joints [49.429, -64.423, 69.517, -0.864, 84.928, 49.502]
  MoveL 457 to (181.42, 208.2, 0) mm, rotated rx 180 ry 0 rz -39.83 deg; joints [49.45, -64.383, 69.46, -0.864, 84.946, 49.523]
  MoveL 458 to (181.73, 208.55, 0) mm, rotated rx 180 ry 0 rz -39.83 deg; joints [49.465, -64.352, 69.416, -0.864, 84.959, 49.538]
  MoveL 459 to (182.02, 208.92, 0) mm, rotated rx 180 ry 0 rz -39.83 deg; joints [49.479, -64.32, 69.37, -0.864, 84.973, 49.552]
  MoveL 460 to (182.29, 209.3, 0) mm, rotated rx 180 ry 0 rz -39.83 deg; joints [49.492, -64.287, 69.323, -0.864, 84.987, 49.565]
  MoveL 461 to (182.55, 209.69, 0) mm, rotated rx -180 ry 0 rz -39.83 deg; joints [49.504, -64.253, 69.274, -0.864, 85.002, 49.577]
  MoveL 462 to (182.73, 210, 0) mm, rotated rx 180 ry 0 rz -39.83 deg; joints [49.513, -64.226, 69.235, -0.864, 85.014, 49.585]
  MoveL 463 to (182.9, 210.32, 0) mm, rotated rx 180 ry 0 rz -39.83 deg; joints [49.521, -64.198, 69.195, -0.864, 85.027, 49.593]
  MoveL 464 to (183.05, 210.65, 0) mm, rotated rx 180 ry 0 rz -39.83 deg; joints [49.529, -64.169, 69.154, -0.864, 85.039, 49.6]
  MoveL 465 to (183.19, 210.99, 0) mm, rotated rx 180 ry 0 rz -39.83 deg; joints [49.535, -64.14, 69.112, -0.864, 85.052, 49.606]
  MoveL 466 to (183.32, 211.4, 0) mm, rotated rx 180 ry 0 rz -39.83 deg; joints [49.541, -64.104, 69.059, -0.864, 85.069, 49.613]
  MoveL 467 to (183.43, 211.83, 0) mm, rotated rx 180 ry 0 rz -39.83 deg; joints [49.547, -64.067, 69.006, -0.863, 85.085, 49.618]
  MoveL 468 to (183.5, 212.26, 0) mm, rotated rx -180 ry 0 rz -39.83 deg; joints [49.55, -64.029, 68.951, -0.863, 85.102, 49.621]
  MoveL 469 to (183.55, 212.69, 0) mm, rotated rx -180 ry 0 rz -39.83 deg; joints [49.553, -63.991, 68.896, -0.863, 85.119, 49.623]
  MoveL 470 to (183.57, 213.04, 0) mm, rotated rx -180 ry 0 rz -39.83 deg; joints [49.554, -63.96, 68.852, -0.863, 85.133, 49.624]
  MoveL 471 to (183.58, 213.39, 0) mm, rotated rx 180 ry 0 rz -39.83 deg; joints [49.554, -63.929, 68.807, -0.863, 85.147, 49.624]
  MoveL 472 to (183.57, 213.74, 0) mm, rotated rx -180 ry 0 rz -39.83 deg; joints [49.554, -63.899, 68.762, -0.863, 85.16, 49.624]
  MoveL 473 to (183.55, 214.09, 0) mm, rotated rx 180 ry 0 rz -39.83 deg; joints [49.554, -63.868, 68.718, -0.863, 85.174, 49.623]
  MoveL 474 to (183.52, 214.42, 0) mm, rotated rx 180 ry 0 rz -39.83 deg; joints [49.553, -63.839, 68.676, -0.863, 85.187, 49.622]
  MoveL 475 to (183.49, 214.74, 0) mm, rotated rx -180 ry 0 rz -39.83 deg; joints [49.551, -63.811, 68.635, -0.863, 85.2, 49.62]
  MoveL 476 to (183.46, 215.07, 0) mm, rotated rx 180 ry 0 rz -39.83 deg; joints [49.55, -63.782, 68.593, -0.863, 85.213, 49.619]
  MoveL 477 to (183.42, 215.39, 0) mm, rotated rx 180 ry 0 rz -39.83 deg; joints [49.548, -63.753, 68.552, -0.863, 85.226, 49.617]
  MoveL 478 to (183.42, 215.39, 0) mm, rotated rx 180 ry 0 rz -39.83 deg; joints [49.548, -63.753, 68.552, -0.863, 85.226, 49.617]
  MoveL 479 to (183.86, 215.85, 0) mm, rotated rx 180 ry 0 rz -39.83 deg; joints [49.569, -63.713, 68.494, -0.863, 85.244, 49.637]
  MoveL 480 to (184.28, 216.32, 0) mm, rotated rx -180 ry 0 rz -39.83 deg; joints [49.589, -63.672, 68.435, -0.863, 85.262, 49.657]
  MoveL 481 to (184.7, 216.8, 0) mm, rotated rx 180 ry 0 rz -39.83 deg; joints [49.608, -63.63, 68.374, -0.863, 85.281, 49.676]
  MoveL 482 to (185.08, 217.3, 0) mm, rotated rx -180 ry 0 rz -39.83 deg; joints [49.627, -63.587, 68.311, -0.863, 85.301, 49.695]
  MoveL 483 to (185.4, 217.75, 0) mm, rotated rx 180 ry 0 rz -39.83 deg; joints [49.642, -63.547, 68.254, -0.863, 85.318, 49.709]
  MoveL 484 to (185.68, 218.22, 0) mm, rotated rx 180 ry 0 rz -39.83 deg; joints [49.655, -63.506, 68.195, -0.863, 85.337, 49.722]
  MoveL 485 to (185.94, 218.71, 0) mm, rotated rx -180 ry 0 rz -39.83 deg; joints [49.667, -63.463, 68.132, -0.863, 85.356, 49.734]
  MoveL 486 to (186.15, 219.21, 0) mm, rotated rx 180 ry 0 rz -39.83 deg; joints [49.677, -63.418, 68.068, -0.863, 85.377, 49.744]
  MoveL 487 to (186.26, 219.52, 0) mm, rotated rx 180 ry 0 rz -39.83 deg; joints [49.682, -63.391, 68.029, -0.863, 85.389, 49.749]
  MoveL 488 to (186.34, 219.83, 0) mm, rotated rx 180 ry 0 rz -39.83 deg; joints [49.687, -63.364, 67.988, -0.863, 85.401, 49.753]
  MoveL 489 to (186.42, 220.15, 0) mm, rotated rx 180 ry 0 rz -39.83 deg; joints [49.69, -63.336, 67.948, -0.863, 85.414, 49.756]
  MoveL 490 to (186.47, 220.47, 0) mm, rotated rx -180 ry 0 rz -39.83 deg; joints [49.693, -63.308, 67.907, -0.863, 85.427, 49.758]
  MoveL 491 to (186.51, 220.83, 0) mm, rotated rx 180 ry 0 rz -39.83 deg; joints [49.695, -63.276, 67.861, -0.863, 85.442, 49.76]
  MoveL 492 to (186.53, 221.19, 0) mm, rotated rx -180 ry 0 rz -39.83 deg; joints [49.696, -63.244, 67.814, -0.863, 85.456, 49.761]
  MoveL 493 to (186.54, 221.55, 0) mm, rotated rx 180 ry 0 rz -39.83 deg; joints [49.696, -63.212, 67.767, -0.863, 85.471, 49.761]
  MoveL 494 to (186.55, 221.91, 0) mm, rotated rx 180 ry 0 rz -39.83 deg; joints [49.697, -63.18, 67.72, -0.863, 85.486, 49.762]
  MoveL 495 to (186.57, 222.18, 0) mm, rotated rx 180 ry 0 rz -39.83 deg; joints [49.698, -63.156, 67.686, -0.863, 85.497, 49.763]
  MoveL 496 to (186.58, 222.45, 0) mm, rotated rx 180 ry 0 rz -39.83 deg; joints [49.699, -63.132, 67.651, -0.863, 85.508, 49.763]
  MoveL 497 to (186.58, 222.72, 0) mm, rotated rx 180 ry 0 rz -39.83 deg; joints [49.699, -63.109, 67.617, -0.863, 85.519, 49.763]
  MoveL 498 to (186.55, 222.98, 0) mm, rotated rx 180 ry 0 rz -39.83 deg; joints [49.698, -63.086, 67.583, -0.863, 85.529, 49.762]
  MoveL 499 to (186.48, 223.29, 0) mm, rotated rx -180 ry 0 rz -39.83 deg; joints [49.694, -63.058, 67.542, -0.863, 85.542, 49.758]
  MoveL 500 to (186.37, 223.59, 0) mm, rotated rx 180 ry 0 rz -39.83 deg; joints [49.689, -63.031, 67.502, -0.863, 85.555, 49.753]
  MoveL 501 to (186.23, 223.89, 0) mm, rotated rx 180 ry 0 rz -39.83 deg; joints [49.683, -63.004, 67.463, -0.863, 85.567, 49.747]
  MoveL 502 to (186.09, 224.19, 0) mm, rotated rx 180 ry 0 rz -39.83 deg; joints [49.676, -62.978, 67.424, -0.863, 85.579, 49.74]
  MoveL 503 to (186.09, 224.19, 0) mm, rotated rx 180 ry 0 rz -39.83 deg; joints [49.676, -62.978, 67.424, -0.863, 85.579, 49.74]
  MoveL 504 to (186.48, 224.74, 0) mm, rotated rx 180 ry 0 rz -39.83 deg; joints [49.695, -62.93, 67.354, -0.863, 85.602, 49.758]
  MoveL 505 to (186.85, 225.29, 0) mm, rotated rx 180 ry 0 rz -39.83 deg; joints [49.712, -62.881, 67.283, -0.863, 85.624, 49.775]
  MoveL 506 to (187.2, 225.86, 0) mm, rotated rx 180 ry 0 rz -39.83 deg; joints [49.729, -62.831, 67.21, -0.863, 85.647, 49.791]
  MoveL 507 to (187.5, 226.45, 0) mm, rotated rx -180 ry 0 rz -39.83 deg; joints [49.743, -62.778, 67.134, -0.863, 85.671, 49.805]
  MoveL 508 to (187.65, 226.82, 0) mm, rotated rx 180 ry 0 rz -39.83 deg; joints [49.75, -62.745, 67.086, -0.863, 85.687, 49.812]
  MoveL 509 to (187.79, 227.2, 0) mm, rotated rx 180 ry 0 rz -39.83 deg; joints [49.756, -62.711, 67.036, -0.863, 85.703, 49.818]
  MoveL 510 to (187.9, 227.59, 0) mm, rotated rx 180 ry 0 rz -39.83 deg; joints [49.762, -62.677, 66.985, -0.863, 85.719, 49.823]
  MoveL 511 to (187.99, 227.99, 0) mm, rotated rx 180 ry 0 rz -39.83 deg; joints [49.766, -62.642, 66.934, -0.863, 85.735, 49.827]
  MoveL 512 to (188.07, 228.44, 0) mm, rotated rx 180 ry 0 rz -39.83 deg; joints [49.77, -62.602, 66.875, -0.863, 85.754, 49.831]
  MoveL 513 to (188.13, 228.89, 0) mm, rotated rx -180 ry 0 rz -39.83 deg; joints [49.773, -62.561, 66.816, -0.863, 85.773, 49.833]
  MoveL 514 to (188.17, 229.35, 0) mm, rotated rx 180 ry 0 rz -39.83 deg; joints [49.775, -62.521, 66.756, -0.863, 85.792, 49.835]
  MoveL 515 to (188.18, 229.8, 0) mm, rotated rx -180 ry 0 rz -39.83 deg; joints [49.776, -62.48, 66.696, -0.863, 85.811, 49.836]
  MoveL 516 to (188.18, 230.2, 0) mm, rotated rx 180 ry 0 rz -39.83 deg; joints [49.776, -62.445, 66.645, -0.862, 85.828, 49.835]
  MoveL 517 to (188.16, 230.59, 0) mm, rotated rx -180 ry 0 rz -39.83 deg; joints [49.775, -62.41, 66.593, -0.862, 85.844, 49.834]
  MoveL 518 to (188.12, 230.98, 0) mm, rotated rx -180 ry 0 rz -39.83 deg; joints [49.773, -62.375, 66.542, -0.862, 85.861, 49.832]
  MoveL 519 to (188.06, 231.36, 0) mm, rotated rx 180 ry 0 rz -39.83 deg; joints [49.77, -62.341, 66.491, -0.862, 85.877, 49.829]
  MoveL 520 to (187.97, 231.74, 0) mm, rotated rx 180 ry 0 rz -39.83 deg; joints [49.766, -62.307, 66.442, -0.862, 85.893, 49.825]
  MoveL 521 to (187.86, 232.1, 0) mm, rotated rx 180 ry 0 rz -39.83 deg; joints [49.761, -62.274, 66.393, -0.862, 85.908, 49.82]
  MoveL 522 to (187.72, 232.46, 0) mm, rotated rx -180 ry 0 rz -39.83 deg; joints [49.755, -62.243, 66.346, -0.862, 85.924, 49.813]
  MoveL 523 to (187.54, 232.8, 0) mm, rotated rx -180 ry 0 rz -39.83 deg; joints [49.747, -62.212, 66.301, -0.862, 85.938, 49.805]
  MoveL 524 to (187.38, 233.05, 0) mm, rotated rx -180 ry 0 rz -39.83 deg; joints [49.739, -62.189, 66.267, -0.862, 85.949, 49.797]
  MoveL 525 to (187.2, 233.3, 0) mm, rotated rx -180 ry 0 rz -39.83 deg; joints [49.731, -62.167, 66.234, -0.862, 85.96, 49.789]
  MoveL 526 to (187.01, 233.54, 0) mm, rotated rx 180 ry 0 rz -39.83 deg; joints [49.723, -62.145, 66.202, -0.862, 85.97, 49.78]
  MoveL 527 to (186.81, 233.78, 0) mm, rotated rx 180 ry 0 rz -39.83 deg; joints [49.714, -62.124, 66.17, -0.862, 85.981, 49.771]
  MoveL 528 to (186.72, 233.9, 0) mm, rotated rx 180 ry 0 rz -39.83 deg; joints [49.709, -62.114, 66.154, -0.862, 85.986, 49.767]
  MoveL 529 to (186.62, 234.02, 0) mm, rotated rx 180 ry 0 rz -39.83 deg; joints [49.705, -62.103, 66.138, -0.862, 85.991, 49.762]
  MoveL 530 to (186.53, 234.13, 0) mm, rotated rx -180 ry 0 rz -39.83 deg; joints [49.701, -62.092, 66.123, -0.862, 85.996, 49.758]
  MoveL 531 to (186.43, 234.25, 0) mm, rotated rx 180 ry 0 rz -39.83 deg; joints [49.696, -62.082, 66.107, -0.862, 86.001, 49.753]
  MoveL 532 to (186.43, 234.25, 0) mm, rotated rx 180 ry 0 rz -39.83 deg; joints [49.696, -62.082, 66.107, -0.862, 86.001, 49.753]
  MoveL 533 to (186.58, 234.43, 0) mm, rotated rx 180 ry 0 rz -39.83 deg; joints [49.703, -62.066, 66.084, -0.862, 86.009, 49.76]
  MoveL 534 to (186.73, 234.61, 0) mm, rotated rx -180 ry 0 rz -39.83 deg; joints [49.71, -62.05, 66.06, -0.862, 86.016, 49.767]
  MoveL 535 to (186.87, 234.79, 0) mm, rotated rx 180 ry 0 rz -39.83 deg; joints [49.717, -62.033, 66.036, -0.862, 86.024, 49.774]
  MoveL 536 to (187.01, 234.98, 0) mm, rotated rx 180 ry 0 rz -39.83 deg; joints [49.723, -62.016, 66.011, -0.862, 86.032, 49.78]
  MoveL 537 to (187.15, 235.22, 0) mm, rotated rx -180 ry 0 rz -39.83 deg; joints [49.73, -61.996, 65.981, -0.862, 86.042, 49.786]
  MoveL 538 to (187.28, 235.46, 0) mm, rotated rx 180 ry 0 rz -39.83 deg; joints [49.736, -61.974, 65.949, -0.862, 86.052, 49.792]
  MoveL 539 to (187.4, 235.71, 0) mm, rotated rx 180 ry 0 rz -39.83 deg; joints [49.741, -61.952, 65.916, -0.862, 86.063, 49.797]
  MoveL 540 to (187.49, 235.97, 0) mm, rotated rx 180 ry 0 rz -39.83 deg; joints [49.746, -61.929, 65.882, -0.862, 86.074, 49.802]
  MoveL 541 to (187.58, 236.27, 0) mm, rotated rx 180 ry 0 rz -39.83 deg; joints [49.75, -61.901, 65.841, -0.862, 86.087, 49.806]
  MoveL 542 to (187.64, 236.59, 0) mm, rotated rx 180 ry 0 rz -39.83 deg; joints [49.753, -61.873, 65.8, -0.862, 86.1, 49.808]
  MoveL 543 to (187.68, 236.9, 0) mm, rotated rx -180 ry 0 rz -39.83 deg; joints [49.755, -61.845, 65.758, -0.862, 86.114, 49.81]
  MoveL 544 to (187.71, 237.22, 0) mm, rotated rx 180 ry 0 rz -39.83 deg; joints [49.756, -61.816, 65.716, -0.862, 86.128, 49.811]
  MoveL 545 to (187.72, 237.55, 0) mm, rotated rx 180 ry 0 rz -39.83 deg; joints [49.757, -61.787, 65.672, -0.862, 86.142, 49.812]
  MoveL 546 to (187.72, 237.88, 0) mm, rotated rx -180 ry 0 rz -39.83 deg; joints [49.757, -61.757, 65.628, -0.862, 86.156, 49.812]
  MoveL 547 to (187.72, 238.21, 0) mm, rotated rx 180 ry 0 rz -39.83 deg; joints [49.757, -61.728, 65.584, -0.862, 86.17, 49.812]
  MoveL 548 to (187.72, 238.54, 0) mm, rotated rx 180 ry 0 rz -39.83 deg; joints [49.757, -61.698, 65.54, -0.862, 86.185, 49.811]
  MoveL 549 to (187.72, 238.93, 0) mm, rotated rx 180 ry 0 rz -39.83 deg; joints [49.757, -61.663, 65.488, -0.862, 86.202, 49.811]
  MoveL 550 to (187.72, 239.32, 0) mm, rotated rx 180 ry 0 rz -39.83 deg; joints [49.757, -61.627, 65.436, -0.862, 86.219, 49.811]
  MoveL 551 to (187.69, 239.71, 0) mm, rotated rx -180 ry 0 rz -39.83 deg; joints [49.756, -61.592, 65.384, -0.862, 86.236, 49.81]
  MoveL 552 to (187.62, 240.09, 0) mm, rotated rx 180 ry 0 rz -39.83 deg; joints [49.753, -61.558, 65.333, -0.862, 86.252, 49.806]
  MoveL 553 to (187.51, 240.41, 0) mm, rotated rx -180 ry 0 rz -39.83 deg; joints [49.748, -61.529, 65.289, -0.862, 86.267, 49.801]
  MoveL 554 to (187.38, 240.73, 0) mm, rotated rx -180 ry 0 rz -39.83 deg; joints [49.742, -61.501, 65.247, -0.862, 86.281, 49.795]
  MoveL 555 to (187.21, 241.03, 0) mm, rotated rx -180 ry 0 rz -39.83 deg; joints [49.735, -61.473, 65.206, -0.862, 86.294, 49.787]
  MoveL 556 to (187.03, 241.33, 0) mm, rotated rx 180 ry 0 rz -39.83 deg; joints [49.726, -61.446, 65.166, -0.862, 86.307, 49.779]
  MoveL 557 to (186.76, 241.73, 0) mm, rotated rx 180 ry 0 rz -39.83 deg; joints [49.714, -61.41, 65.111, -0.862, 86.325, 49.766]
  MoveL 558 to (186.46, 242.12, 0) mm, rotated rx -180 ry 0 rz -39.83 deg; joints [49.701, -61.375, 65.058, -0.862, 86.343, 49.753]
  MoveL 559 to (186.14, 242.48, 0) mm, rotated rx 180 ry 0 rz -39.83 deg; joints [49.686, -61.342, 65.009, -0.862, 86.359, 49.738]
  MoveL 560 to (185.79, 242.81, 0) mm, rotated rx 180 ry 0 rz -39.83 deg; joints [49.67, -61.312, 64.964, -0.862, 86.374, 49.722]
  MoveL 561 to (185.55, 243.01, 0) mm, rotated rx -180 ry 0 rz -39.83 deg; joints [49.659, -61.294, 64.937, -0.862, 86.383, 49.711]
  MoveL 562 to (185.29, 243.19, 0) mm, rotated rx -180 ry 0 rz -39.83 deg; joints [49.648, -61.278, 64.912, -0.862, 86.391, 49.699]
  MoveL 563 to (185.03, 243.35, 0) mm, rotated rx 180 ry 0 rz -39.83 deg; joints [49.636, -61.262, 64.889, -0.862, 86.398, 49.687]
  MoveL 564 to (184.75, 243.5, 0) mm, rotated rx -180 ry 0 rz -39.83 deg; joints [49.623, -61.249, 64.869, -0.862, 86.405, 49.674]
  MoveL 565 to (184.45, 243.64, 0) mm, rotated rx -180 ry 0 rz -39.83 deg; joints [49.609, -61.236, 64.849, -0.862, 86.412, 49.66]
  MoveL 566 to (184.13, 243.77, 0) mm, rotated rx -180 ry 0 rz -39.83 deg; joints [49.595, -61.224, 64.831, -0.862, 86.418, 49.646]
  MoveL 567 to (183.81, 243.87, 0) mm, rotated rx -180 ry 0 rz -39.83 deg; joints [49.58, -61.215, 64.817, -0.862, 86.422, 49.631]
  MoveL 568 to (183.48, 243.95, 0) mm, rotated rx 180 ry 0 rz -39.83 deg; joints [49.565, -61.207, 64.805, -0.862, 86.426, 49.616]
  MoveL 569 to (183.15, 244.01, 0) mm, rotated rx 180 ry 0 rz -39.83 deg; joints [49.55, -61.202, 64.797, -0.862, 86.429, 49.601]
  MoveL 570 to (182.83, 244.04, 0) mm, rotated rx 180 ry 0 rz -39.83 deg; joints [49.535, -61.198, 64.791, -0.862, 86.431, 49.586]
  MoveL 571 to (182.5, 244.07, 0) mm, rotated rx 180 ry 0 rz -39.83 deg; joints [49.52, -61.196, 64.786, -0.862, 86.433, 49.571]
  MoveL 572 to (182.17, 244.09, 0) mm, rotated rx 180 ry 0 rz -39.83 deg; joints [49.505, -61.194, 64.783, -0.862, 86.434, 49.556]
  MoveL 573 to (181.73, 244.1, 0) mm, rotated rx 180 ry 0 rz -39.83 deg; joints [49.486, -61.192, 64.78, -0.862, 86.435, 49.536]
  MoveL 574 to (181.3, 244.1, 0) mm, rotated rx 180 ry 0 rz -39.83 deg; joints [49.466, -61.192, 64.779, -0.862, 86.435, 49.516]
  MoveL 575 to (180.87, 244.09, 0) mm, rotated rx -180 ry 0 rz -39.83 deg; joints [49.446, -61.193, 64.78, -0.862, 86.435, 49.497]
  MoveL 576 to (180.44, 244.05, 0) mm, rotated rx -180 ry 0 rz -39.83 deg; joints [49.426, -61.195, 64.783, -0.862, 86.434, 49.477]
  MoveL 577 to (180.19, 244.02, 0) mm, rotated rx 180 ry 0 rz -39.83 deg; joints [49.415, -61.198, 64.787, -0.862, 86.433, 49.466]
  MoveL 578 to (179.94, 243.99, 0) mm, rotated rx 180 ry 0 rz -39.83 deg; joints [49.404, -61.2, 64.79, -0.862, 86.432, 49.454]
  MoveL 579 to (179.69, 243.95, 0) mm, rotated rx -180 ry 0 rz -39.83 deg; joints [49.392, -61.204, 64.795, -0.862, 86.43, 49.443]
  MoveL 580 to (179.44, 243.91, 0) mm, rotated rx -180 ry 0 rz -39.83 deg; joints [49.381, -61.207, 64.799, -0.862, 86.429, 49.431]
  MoveL 581 to (179.31, 243.9, 0) mm, rotated rx 180 ry 0 rz -39.83 deg; joints [49.375, -61.208, 64.801, -0.862, 86.428, 49.425]
  MoveL 582 to (179.18, 243.88, 0) mm, rotated rx 180 ry 0 rz -39.83 deg; joints [49.369, -61.209, 64.803, -0.862, 86.428, 49.42]
  MoveL 583 to (179.05, 243.86, 0) mm, rotated rx -180 ry 0 rz -39.83 deg; joints [49.363, -61.211, 64.805, -0.862, 86.427, 49.414]
  MoveL 584 to (178.92, 243.85, 0) mm, rotated rx 180 ry 0 rz -39.83 deg; joints [49.357, -61.212, 64.807, -0.862, 86.427, 49.408]
  MoveL 585 to (178.92, 243.85, 0) mm, rotated rx 180 ry 0 rz -39.83 deg; joints [49.357, -61.212, 64.807, -0.862, 86.427, 49.408]
  MoveL 586 to (178.79, 244.05, 0) mm, rotated rx 180 ry 0 rz -39.83 deg; joints [49.351, -61.193, 64.779, -0.862, 86.436, 49.402]
  MoveL 587 to (178.65, 244.26, 0) mm, rotated rx 180 ry 0 rz -39.83 deg; joints [49.345, -61.175, 64.75, -0.862, 86.445, 49.395]
  MoveL 588 to (178.52, 244.46, 0) mm, rotated rx 180 ry 0 rz -39.83 deg; joints [49.339, -61.156, 64.722, -0.862, 86.454, 49.389]
  MoveL 589 to (178.38, 244.66, 0) mm, rotated rx -180 ry 0 rz -39.83 deg; joints [49.333, -61.138, 64.695, -0.862, 86.464, 49.383]
  MoveL 590 to (178.19, 244.93, 0) mm, rotated rx 180 ry 0 rz -39.83 deg; joints [49.324, -61.113, 64.657, -0.862, 86.476, 49.374]
  MoveL 591 to (177.99, 245.2, 0) mm, rotated rx 180 ry 0 rz -39.83 deg; joints [49.315, -61.089, 64.621, -0.862, 86.488, 49.365]
  MoveL 592 to (177.78, 245.46, 0) mm, rotated rx 180 ry 0 rz -39.83 deg; joints [49.306, -61.065, 64.585, -0.862, 86.5, 49.356]
  MoveL 593 to (177.57, 245.72, 0) mm, rotated rx 180 ry 0 rz -39.83 deg; joints [49.296, -61.041, 64.55, -0.862, 86.512, 49.346]
  MoveL 594 to (177.38, 245.92, 0) mm, rotated rx 180 ry 0 rz -39.83 deg; joints [49.288, -61.022, 64.521, -0.862, 86.521, 49.337]
  MoveL 595 to (177.19, 246.12, 0) mm, rotated rx -180 ry 0 rz -39.83 deg; joints [49.279, -61.004, 64.494, -0.862, 86.53, 49.329]
  MoveL 596 to (176.99, 246.3, 0) mm, rotated rx 180 ry 0 rz -39.83 deg; joints [49.27, -60.988, 64.469, -0.862, 86.538, 49.319]
  MoveL 597 to (176.77, 246.46, 0) mm, rotated rx -180 ry 0 rz -39.83 deg; joints [49.261, -60.973, 64.447, -0.862, 86.546, 49.309]
  MoveL 598 to (176.44, 246.65, 0) mm, rotated rx 180 ry 0 rz -39.83 deg; joints [49.246, -60.956, 64.421, -0.862, 86.555, 49.294]
  MoveL 599 to (176.08, 246.79, 0) mm, rotated rx 180 ry 0 rz -39.83 deg; joints [49.229, -60.942, 64.4, -0.862, 86.562, 49.278]
  MoveL 600 to (175.71, 246.91, 0) mm, rotated rx 180 ry 0 rz -39.83 deg; joints [49.213, -60.931, 64.383, -0.862, 86.567, 49.261]
  MoveL 601 to (175.34, 247, 0) mm, rotated rx 180 ry 0 rz -39.83 deg; joints [49.196, -60.922, 64.369, -0.862, 86.572, 49.244]
  MoveL 602 to (175.08, 247.06, 0) mm, rotated rx 180 ry 0 rz -39.83 deg; joints [49.184, -60.916, 64.36, -0.862, 86.575, 49.232]
  MoveL 603 to (174.82, 247.11, 0) mm, rotated rx 180 ry 0 rz -39.83 deg; joints [49.172, -60.911, 64.352, -0.862, 86.578, 49.22]
  MoveL 604 to (174.56, 247.16, 0) mm, rotated rx -180 ry 0 rz -39.83 deg; joints [49.16, -60.906, 64.345, -0.862, 86.58, 49.209]
  MoveL 605 to (174.3, 247.2, 0) mm, rotated rx 180 ry 0 rz -39.83 deg; joints [49.148, -60.902, 64.338, -0.862, 86.582, 49.197]
  MoveL 606 to (173.79, 247.27, 0) mm, rotated rx 180 ry 0 rz -39.83 deg; joints [49.125, -60.895, 64.326, -0.862, 86.586, 49.174]
  MoveL 607 to (173.28, 247.33, 0) mm, rotated rx 180 ry 0 rz -39.83 deg; joints [49.102, -60.889, 64.317, -0.862, 86.589, 49.15]
  MoveL 608 to (172.77, 247.37, 0) mm, rotated rx -180 ry 0 rz -39.83 deg; joints [49.079, -60.885, 64.309, -0.862, 86.592, 49.127]
  MoveL 609 to (172.26, 247.4, 0) mm, rotated rx -180 ry 0 rz -39.83 deg; joints [49.056, -60.881, 64.303, -0.862, 86.594, 49.104]
  MoveL 610 to (171.69, 247.44, 0) mm, rotated rx -180 ry 0 rz -39.83 deg; joints [49.03, -60.877, 64.297, -0.862, 86.596, 49.078]
  MoveL 611 to (171.12, 247.46, 0) mm, rotated rx 180 ry 0 rz -39.83 deg; joints [49.004, -60.874, 64.291, -0.862, 86.598, 49.052]
  MoveL 612 to (170.56, 247.47, 0) mm, rotated rx 180 ry 0 rz -39.83 deg; joints [48.978, -60.872, 64.287, -0.862, 86.6, 49.026]
  MoveL 613 to (169.99, 247.47, 0) mm, rotated rx 180 ry 0 rz -39.83 deg; joints [48.952, -60.871, 64.285, -0.862, 86.601, 49]
  MoveL 614 to (169.4, 247.46, 0) mm, rotated rx 180 ry 0 rz -39.83 deg; joints [48.925, -60.871, 64.284, -0.862, 86.601, 48.973]
  MoveL 615 to (168.81, 247.44, 0) mm, rotated rx 180 ry 0 rz -39.83 deg; joints [48.898, -60.871, 64.285, -0.862, 86.601, 48.946]
  MoveL 616 to (168.21, 247.41, 0) mm, rotated rx -180 ry 0 rz -39.83 deg; joints [48.872, -60.873, 64.286, -0.862, 86.6, 48.92]
  MoveL 617 to (167.62, 247.38, 0) mm, rotated rx 180 ry 0 rz -39.83 deg; joints [48.845, -60.875, 64.288, -0.862, 86.6, 48.893]
  MoveL 618 to (167.62, 247.38, 0) mm, rotated rx 180 ry 0 rz -39.83 deg; joints [48.845, -60.875, 64.288, -0.862, 86.6, 48.893]
  MoveL 619 to (167.57, 247.54, 0) mm, rotated rx 180 ry 0 rz -39.83 deg; joints [48.842, -60.86, 64.266, -0.862, 86.607, 48.89]
  MoveL 620 to (167.52, 247.7, 0) mm, rotated rx 180 ry 0 rz -39.83 deg; joints [48.84, -60.845, 64.243, -0.862, 86.615, 48.888]
  MoveL 621 to (167.45, 247.86, 0) mm, rotated rx 180 ry 0 rz -39.83 deg; joints [48.837, -60.831, 64.222, -0.862, 86.622, 48.885]
  MoveL 622 to (167.37, 248.01, 0) mm, rotated rx -180 ry 0 rz -39.83 deg; joints [48.834, -60.817, 64.201, -0.862, 86.629, 48.881]
  MoveL 623 to (167.27, 248.16, 0) mm, rotated rx 180 ry 0 rz -39.83 deg; joints [48.829, -60.803, 64.181, -0.862, 86.636, 48.877]
  MoveL 624 to (167.16, 248.3, 0) mm, rotated rx -180 ry 0 rz -39.83 deg; joints [48.824, -60.79, 64.161, -0.862, 86.642, 48.872]
  MoveL 625 to (167.03, 248.43, 0) mm, rotated rx 180 ry 0 rz -39.83 deg; joints [48.819, -60.778, 64.142, -0.862, 86.648, 48.866]
  MoveL 626 to (166.89, 248.56, 0) mm, rotated rx -180 ry 0 rz -39.83 deg; joints [48.812, -60.766, 64.125, -0.862, 86.654, 48.86]
  MoveL 627 to (166.69, 248.74, 0) mm, rotated rx -180 ry 0 rz -39.83 deg; joints [48.803, -60.749, 64.099, -0.862, 86.663, 48.851]
  MoveL 628 to (166.48, 248.91, 0) mm, rotated rx 180 ry 0 rz -39.83 deg; joints [48.794, -60.734, 64.075, -0.862, 86.671, 48.841]
  MoveL 629 to (166.26, 249.06, 0) mm, rotated rx -180 ry 0 rz -39.83 deg; joints [48.784, -60.719, 64.053, -0.862, 86.678, 48.831]
  MoveL 630 to (166.03, 249.2, 0) mm, rotated rx 180 ry 0 rz -39.83 deg; joints [48.774, -60.706, 64.034, -0.862, 86.685, 48.821]
  MoveL 631 to (165.78, 249.32, 0) mm, rotated rx -180 ry 0 rz -39.83 deg; joints [48.763, -60.695, 64.016, -0.862, 86.691, 48.809]
  MoveL 632 to (165.51, 249.42, 0) mm, rotated rx -180 ry 0 rz -39.83 deg; joints [48.751, -60.685, 64.001, -0.862, 86.696, 48.797]
  MoveL 633 to (165.23, 249.51, 0) mm, rotated rx 180 ry 0 rz -39.83 deg; joints [48.738, -60.676, 63.988, -0.862, 86.7, 48.785]
  MoveL 634 to (164.95, 249.59, 0) mm, rotated rx 180 ry 0 rz -39.83 deg; joints [48.726, -60.668, 63.975, -0.862, 86.704, 48.772]
  MoveL 635 to (164.59, 249.7, 0) mm, rotated rx 180 ry 0 rz -39.83 deg; joints [48.709, -60.658, 63.96, -0.862, 86.71, 48.755]
  MoveL 636 to (164.22, 249.79, 0) mm, rotated rx 180 ry 0 rz -39.83 deg; joints [48.692, -60.648, 63.945, -0.862, 86.715, 48.739]
  MoveL 637 to (163.85, 249.88, 0) mm, rotated rx -180 ry 0 rz -39.83 deg; joints [48.676, -60.64, 63.932, -0.862, 86.719, 48.722]
  MoveL 638 to (163.48, 249.94, 0) mm, rotated rx 180 ry 0 rz -39.83 deg; joints [48.659, -60.633, 63.92, -0.862, 86.723, 48.705]
  MoveL 639 to (162.96, 250.01, 0) mm, rotated rx 180 ry 0 rz -39.83 deg; joints [48.635, -60.626, 63.909, -0.862, 86.727, 48.681]
  MoveL 640 to (162.43, 250.04, 0) mm, rotated rx 180 ry 0 rz -39.83 deg; joints [48.611, -60.622, 63.903, -0.862, 86.729, 48.657]
  MoveL 641 to (161.9, 250.04, 0) mm, rotated rx 180 ry 0 rz -39.83 deg; joints [48.587, -60.621, 63.9, -0.862, 86.73, 48.633]
  MoveL 642 to (161.37, 250.01, 0) mm, rotated rx 180 ry 0 rz -39.83 deg; joints [48.563, -60.622, 63.901, -0.862, 86.73, 48.609]
  MoveL 643 to (160.95, 249.97, 0) mm, rotated rx 180 ry 0 rz -39.83 deg; joints [48.544, -60.624, 63.904, -0.862, 86.729, 48.59]
  MoveL 644 to (160.53, 249.93, 0) mm, rotated rx -180 ry 0 rz -39.83 deg; joints [48.525, -60.627, 63.909, -0.862, 86.727, 48.571]
  MoveL 645 to (160.11, 249.87, 0) mm, rotated rx 180 ry 0 rz -39.83 deg; joints [48.506, -60.631, 63.914, -0.862, 86.726, 48.552]
  MoveL 646 to (159.69, 249.81, 0) mm, rotated rx 180 ry 0 rz -39.83 deg; joints [48.487, -60.636, 63.92, -0.862, 86.724, 48.533]
  MoveL 647 to (159.69, 249.81, 0) mm, rotated rx 180 ry 0 rz -39.83 deg; joints [48.487, -60.636, 63.92, -0.862, 86.724, 48.533]
  MoveL 648 to (159.6, 249.96, 0) mm, rotated rx 180 ry 0 rz -39.83 deg; joints [48.483, -60.622, 63.9, -0.862, 86.73, 48.529]
  MoveL 649 to (159.5, 250.09, 0) mm, rotated rx 180 ry 0 rz -39.83 deg; joints [48.479, -60.61, 63.88, -0.862, 86.737, 48.524]
  MoveL 650 to (159.4, 250.23, 0) mm, rotated rx 180 ry 0 rz -39.83 deg; joints [48.474, -60.597, 63.861, -0.862, 86.743, 48.52]
  MoveL 651 to (159.3, 250.36, 0) mm, rotated rx 180 ry 0 rz -39.83 deg; joints [48.47, -60.585, 63.843, -0.862, 86.75, 48.515]
  MoveL 652 to (159.11, 250.57, 0) mm, rotated rx -180 ry 0 rz -39.83 deg; joints [48.461, -60.565, 63.813, -0.862, 86.759, 48.507]
  MoveL 653 to (158.9, 250.76, 0) mm, rotated rx 180 ry 0 rz -39.83 deg; joints [48.452, -60.547, 63.786, -0.862, 86.769, 48.497]
  MoveL 654 to (158.67, 250.93, 0) mm, rotated rx 180 ry 0 rz -39.83 deg; joints [48.442, -60.531, 63.761, -0.862, 86.777, 48.487]
  MoveL 655 to (158.44, 251.09, 0) mm, rotated rx 180 ry 0 rz -39.83 deg; joints [48.432, -60.516, 63.739, -0.862, 86.784, 48.477]
  MoveL 656 to (158.09, 251.28, 0) mm, rotated rx 180 ry 0 rz -39.83 deg; joints [48.416, -60.498, 63.711, -0.862, 86.794, 48.461]
  MoveL 657 to (157.72, 251.44, 0) mm, rotated rx 180 ry 0 rz -39.83 deg; joints [48.4, -60.483, 63.688, -0.862, 86.802, 48.444]
  MoveL 658 to (157.35, 251.58, 0) mm, rotated rx 180 ry 0 rz -39.83 deg; joints [48.383, -60.469, 63.667, -0.862, 86.809, 48.427]
  MoveL 659 to (156.97, 251.7, 0) mm, rotated rx 180 ry 0 rz -39.83 deg; joints [48.366, -60.456, 63.647, -0.862, 86.815, 48.41]
  MoveL 660 to (156.61, 251.82, 0) mm, rotated rx 180 ry 0 rz -39.83 deg; joints [48.35, -60.445, 63.629, -0.862, 86.821, 48.394]
  MoveL 661 to (156.26, 251.93, 0) mm, rotated rx 180 ry 0 rz -39.83 deg; joints [48.334, -60.434, 63.613, -0.862, 86.827, 48.378]
  MoveL 662 to (155.9, 252.02, 0) mm, rotated rx 180 ry 0 rz -39.83 deg; joints [48.318, -60.425, 63.598, -0.862, 86.832, 48.362]
  MoveL 663 to (155.54, 252.08, 0) mm, rotated rx 180 ry 0 rz -39.83 deg; joints [48.301, -60.418, 63.588, -0.862, 86.835, 48.346]
  MoveL 664 to (155.08, 252.11, 0) mm, rotated rx 180 ry 0 rz -39.83 deg; joints [48.28, -60.414, 63.581, -0.862, 86.838, 48.325]
  MoveL 665 to (154.61, 252.09, 0) mm, rotated rx 180 ry 0 rz -39.83 deg; joints [48.259, -60.414, 63.58, -0.862, 86.838, 48.304]
  MoveL 666 to (154.15, 252.04, 0) mm, rotated rx -180 ry 0 rz -39.83 deg; joints [48.238, -60.417, 63.585, -0.862, 86.837, 48.283]
  MoveL 667 to (153.69, 251.97, 0) mm, rotated rx 180 ry 0 rz -39.83 deg; joints [48.217, -60.423, 63.593, -0.862, 86.834, 48.262]
  MoveL 668 to (153.17, 251.86, 0) mm, rotated rx 180 ry 0 rz -39.83 deg; joints [48.194, -60.431, 63.604, -0.862, 86.83, 48.238]
  MoveL 669 to (152.66, 251.74, 0) mm, rotated rx 180 ry 0 rz -39.83 deg; joints [48.17, -60.441, 63.618, -0.862, 86.826, 48.215]
  MoveL 670 to (152.15, 251.6, 0) mm, rotated rx -180 ry 0 rz -39.83 deg; joints [48.147, -60.451, 63.633, -0.862, 86.821, 48.192]
  MoveL 671 to (151.64, 251.46, 0) mm, rotated rx -180 ry 0 rz -39.83 deg; joints [48.124, -60.463, 63.65, -0.862, 86.815, 48.168]
  MoveL 672 to (151.08, 251.3, 0) mm, rotated rx 180 ry 0 rz -39.83 deg; joints [48.098, -60.476, 63.669, -0.862, 86.809, 48.143]
  MoveL 673 to (150.52, 251.14, 0) mm, rotated rx 180 ry 0 rz -39.83 deg; joints [48.072, -60.489, 63.688, -0.862, 86.803, 48.117]
  MoveL 674 to (149.95, 250.97, 0) mm, rotated rx -180 ry 0 rz -39.83 deg; joints [48.046, -60.502, 63.707, -0.862, 86.796, 48.091]
  MoveL 675 to (149.39, 250.8, 0) mm, rotated rx 180 ry 0 rz -39.83 deg; joints [48.021, -60.516, 63.727, -0.862, 86.79, 48.066]
  MoveL 676 to (149.39, 250.8, 0) mm, rotated rx 180 ry 0 rz -39.83 deg; joints [48.021, -60.516, 63.727, -0.862, 86.79, 48.066]
  MoveL 677 to (149.09, 251.08, 0) mm, rotated rx 180 ry 0 rz -39.83 deg; joints [48.007, -60.489, 63.686, -0.862, 86.804, 48.052]
  MoveL 678 to (148.77, 251.35, 0) mm, rotated rx -180 ry 0 rz -39.83 deg; joints [47.993, -60.463, 63.647, -0.862, 86.817, 48.038]
  MoveL 679 to (148.45, 251.61, 0) mm, rotated rx 180 ry 0 rz -39.83 deg; joints [47.979, -60.439, 63.61, -0.862, 86.829, 48.024]
  MoveL 680 to (148.1, 251.83, 0) mm, rotated rx 180 ry 0 rz -39.83 deg; joints [47.964, -60.418, 63.578, -0.862, 86.84, 48.008]
  MoveL 681 to (147.83, 251.97, 0) mm, rotated rx 180 ry 0 rz -39.83 deg; joints [47.952, -60.404, 63.557, -0.862, 86.847, 47.996]
  MoveL 682 to (147.54, 252.09, 0) mm, rotated rx 180 ry 0 rz -39.83 deg; joints [47.939, -60.392, 63.539, -0.862, 86.853, 47.983]
  MoveL 683 to (147.24, 252.18, 0) mm, rotated rx 180 ry 0 rz -39.83 deg; joints [47.926, -60.383, 63.524, -0.862, 86.858, 47.97]
  MoveL 684 to (146.94, 252.24, 0) mm, rotated rx 180 ry 0 rz -39.83 deg; joints [47.912, -60.376, 63.513, -0.862, 86.862, 47.956]
  MoveL 685 to (146.49, 252.3, 0) mm, rotated rx -180 ry 0 rz -39.83 deg; joints [47.892, -60.37, 63.503, -0.862, 86.865, 47.936]
  MoveL 686 to (146.04, 252.3, 0) mm, rotated rx 180 ry 0 rz -39.83 deg; joints [47.871, -60.367, 63.499, -0.862, 86.867, 47.915]
  MoveL 687 to (145.58, 252.27, 0) mm, rotated rx -180 ry 0 rz -39.83 deg; joints [47.85, -60.368, 63.5, -0.862, 86.866, 47.894]
  MoveL 688 to (145.12, 252.22, 0) mm, rotated rx 180 ry 0 rz -39.83 deg; joints [47.83, -60.371, 63.504, -0.862, 86.865, 47.873]
  MoveL 689 to (144.65, 252.15, 0) mm, rotated rx 180 ry 0 rz -39.83 deg; joints [47.808, -60.376, 63.511, -0.862, 86.863, 47.852]
  MoveL 690 to (144.18, 252.07, 0) mm, rotated rx 180 ry 0 rz -39.83 deg; joints [47.787, -60.382, 63.519, -0.862, 86.861, 47.831]
  MoveL 691 to (143.72, 251.97, 0) mm, rotated rx 180 ry 0 rz -39.83 deg; joints [47.766, -60.389, 63.529, -0.862, 86.857, 47.81]
  MoveL 692 to (143.26, 251.85, 0) mm, rotated rx 180 ry 0 rz -39.83 deg; joints [47.745, -60.399, 63.543, -0.862, 86.853, 47.789]
  MoveL 693 to (142.8, 251.7, 0) mm, rotated rx -180 ry 0 rz -39.83 deg; joints [47.723, -60.41, 63.56, -0.862, 86.847, 47.767]
  MoveL 694 to (142.34, 251.54, 0) mm, rotated rx 180 ry 0 rz -39.83 deg; joints [47.702, -60.424, 63.579, -0.862, 86.841, 47.746]
  MoveL 695 to (141.88, 251.36, 0) mm, rotated rx -180 ry 0 rz -39.83 deg; joints [47.681, -60.438, 63.601, -0.862, 86.834, 47.725]
  MoveL 696 to (141.42, 251.17, 0) mm, rotated rx 180 ry 0 rz -39.83 deg; joints [47.66, -60.453, 63.623, -0.862, 86.826, 47.704]
  MoveL 697 to (140.87, 250.94, 0) mm, rotated rx 180 ry 0 rz -39.83 deg; joints [47.634, -60.472, 63.65, -0.862, 86.817, 47.679]
  MoveL 698 to (140.33, 250.71, 0) mm, rotated rx 180 ry 0 rz -39.83 deg; joints [47.609, -60.491, 63.678, -0.862, 86.808, 47.654]
  MoveL 699 to (139.78, 250.48, 0) mm, rotated rx -180 ry 0 rz -39.83 deg; joints [47.584, -60.51, 63.705, -0.862, 86.799, 47.629]
  MoveL 700 to (139.23, 250.25, 0) mm, rotated rx -180 ry 0 rz -39.83 deg; joints [47.558, -60.529, 63.733, -0.862, 86.79, 47.603]
  MoveL 701 to (139.23, 250.25, 0) mm, rotated rx -180 ry 0 rz -39.83 deg; joints [47.558, -60.529, 63.733, -0.862, 86.79, 47.603]
  MoveL 702 to (138.91, 250.41, 0) mm, rotated rx 180 ry 0 rz -39.83 deg; joints [47.544, -60.513, 63.709, -0.862, 86.798, 47.589]
  MoveL 703 to (138.58, 250.56, 0) mm, rotated rx 180 ry 0 rz -39.83 deg; joints [47.53, -60.498, 63.686, -0.862, 86.806, 47.574]
  MoveL 704 to (138.25, 250.7, 0) mm, rotated rx 180 ry 0 rz -39.83 deg; joints [47.515, -60.484, 63.665, -0.862, 86.813, 47.56]
  MoveL 705 to (137.92, 250.82, 0) mm, rotated rx 180 ry 0 rz -39.83 deg; joints [47.5, -60.472, 63.645, -0.862, 86.819, 47.545]
  MoveL 706 to (137.61, 250.91, 0) mm, rotated rx 180 ry 0 rz -39.83 deg; joints [47.486, -60.462, 63.631, -0.862, 86.824, 47.531]
  MoveL 707 to (137.3, 250.98, 0) mm, rotated rx 180 ry 0 rz -39.83 deg; joints [47.472, -60.455, 63.619, -0.862, 86.828, 47.517]
  MoveL 708 to (136.98, 251.03, 0) mm, rotated rx 180 ry 0 rz -39.83 deg; joints [47.458, -60.449, 63.61, -0.862, 86.831, 47.503]
  MoveL 709 to (136.67, 251.06, 0) mm, rotated rx 180 ry 0 rz -39.83 deg; joints [47.444, -60.444, 63.603, -0.862, 86.834, 47.488]
  MoveL 710 to (136.36, 251.08, 0) mm, rotated rx 180 ry 0 rz -39.83 deg; joints [47.43, -60.442, 63.599, -0.862, 86.835, 47.474]
  MoveL 711 to (136.05, 251.08, 0) mm, rotated rx 180 ry 0 rz -39.83 deg; joints [47.416, -60.44, 63.596, -0.862, 86.836, 47.461]
  MoveL 712 to (135.75, 251.06, 0) mm, rotated rx 180 ry 0 rz -39.83 deg; joints [47.402, -60.44, 63.596, -0.862, 86.836, 47.447]
  MoveL 713 to (135.44, 251.04, 0) mm, rotated rx 180 ry 0 rz -39.83 deg; joints [47.388, -60.441, 63.597, -0.862, 86.836, 47.433]
  MoveL 714 to (135.08, 251, 0) mm, rotated rx 180 ry 0 rz -39.83 deg; joints [47.372, -60.443, 63.6, -0.862, 86.835, 47.416]
  MoveL 715 to (134.72, 250.94, 0) mm, rotated rx 180 ry 0 rz -39.83 deg; joints [47.356, -60.447, 63.605, -0.862, 86.833, 47.4]
  MoveL 716 to (134.37, 250.87, 0) mm, rotated rx 180 ry 0 rz -39.83 deg; joints [47.339, -60.452, 63.612, -0.862, 86.831, 47.384]
  MoveL 717 to (134.02, 250.78, 0) mm, rotated rx 180 ry 0 rz -39.83 deg; joints [47.323, -60.459, 63.622, -0.862, 86.828, 47.368]
  MoveL 718 to (133.61, 250.65, 0) mm, rotated rx 180 ry 0 rz -39.83 deg; joints [47.305, -60.469, 63.636, -0.862, 86.823, 47.349]
  MoveL 719 to (133.21, 250.49, 0) mm, rotated rx 180 ry 0 rz -39.83 deg; joints [47.286, -60.481, 63.654, -0.862, 86.817, 47.331]
  MoveL 720 to (132.82, 250.31, 0) mm, rotated rx 180 ry 0 rz -39.83 deg; joints [47.268, -60.496, 63.675, -0.862, 86.81, 47.313]
  MoveL 721 to (132.44, 250.12, 0) mm, rotated rx -180 ry 0 rz -39.83 deg; joints [47.25, -60.512, 63.699, -0.862, 86.802, 47.295]
  MoveL 722 to (131.93, 249.82, 0) mm, rotated rx 180 ry 0 rz -39.83 deg; joints [47.226, -60.536, 63.735, -0.862, 86.79, 47.271]
  MoveL 723 to (131.42, 249.51, 0) mm, rotated rx 180 ry 0 rz -39.83 deg; joints [47.203, -60.563, 63.775, -0.862, 86.777, 47.248]
  MoveL 724 to (130.93, 249.17, 0) mm, rotated rx 180 ry 0 rz -39.83 deg; joints [47.179, -60.591, 63.816, -0.862, 86.764, 47.225]
  MoveL 725 to (130.44, 248.83, 0) mm, rotated rx 180 ry 0 rz -39.83 deg; joints [47.156, -60.62, 63.859, -0.862, 86.749, 47.202]
  MoveL 726 to (130.44, 248.83, 0) mm, rotated rx 180 ry 0 rz -39.83 deg; joints [47.156, -60.62, 63.859, -0.862, 86.749, 47.202]
  MoveL 727 to (130.24, 248.89, 0) mm, rotated rx 180 ry 0 rz -39.83 deg; joints [47.148, -60.614, 63.849, -0.862, 86.753, 47.193]
  MoveL 728 to (130.05, 248.95, 0) mm, rotated rx 180 ry 0 rz -39.83 deg; joints [47.139, -60.608, 63.84, -0.862, 86.756, 47.184]
  MoveL 729 to (129.85, 249, 0) mm, rotated rx 180 ry 0 rz -39.83 deg; joints [47.13, -60.602, 63.831, -0.862, 86.759, 47.175]
